    M_KRONOTECH_SRL : UINT := 814; (* Manufacturer: Kronotech Srl (formerly Soltec Soluzioni Tecnologiche Srl) | Location: Basaldella *)
    M_FLIR_SYSTEMS : UINT := 815; (* Manufacturer: FLIR Systems, Inc. | Location: Wilsonville, OR USA - 2017-04-21 *)
    M_UNISTRONG : UINT := 816; (* Manufacturer: UniStrong | Location: Beijing, China - 2017-04-21 *)
    M_TE_CONNECTIVITY_SENSOR_SOLUTIONS : UINT := 817; (* Manufacturer: TE Connectivity Sensor Solutions | Location: Dormund, Germany - 2017-04-21 *)
    M_HGNSS : UINT := 818; (* Manufacturer: HGNSS | Location: Scottsdale, AZ USA - 2017-04-21 *)
    M_PRECO_ELECTRONICS : UINT := 819; (* Manufacturer: Preco Electronics | Location: Boise, ID USA - 2017-04-30 *)
    M_DIALOGIKA_GESELLSCHAFT_FUER_ANGEWANDTE_INFORMATIK_MBH : UINT := 820; (* Manufacturer: DIaLOGIKa Gesellschaft fuer angewandte Informatik mbH | Location: Saarbruecken, *)
    M_THORSEN_TEKNIK : UINT := 821; (* Manufacturer: Thorsen Teknik A/S | Location: Farsø, Denmark - 2017-05-01 *)
    M_BREN_TRONICS : UINT := 822; (* Manufacturer: Bren-Tronics, Inc. | Location: Commack, NY USA - 2017-05-04 *)
    M_ACEINNA : UINT := 823; (* Manufacturer: ACEINNA, Inc (formerly MEMSIC, Inc) | Location: Andover, MA USA - 2017-09-03 *)
    M_UNDHEIM_SYSTEMS : UINT := 824; (* Manufacturer: Undheim Systems AS | Location: Egersund, Norway - 2017-05-04 *)
    M_BPW_HUNG_RIA : UINT := 825; (* Manufacturer: BPW Hungária | Location: Szombathely, Hungary - 2017-05-04 *)
    M_LEWMAR_MARINE : UINT := 826; (* Manufacturer: Lewmar Marine Inc | Location: Guilford, CT USA - 2017-05-05 *)
    M_INMATIX_TECHNOLOGY_GROUP : UINT := 827; (* Manufacturer: INmatix Technology Group Ltd | Location: Hattem, The Netherlands - 2017-05-11 *)
    M_AGRIBRINK : UINT := 828; (* Manufacturer: AgriBrink Inc. | Location: Moorefield, ON Canada - 2017-05-21 *)
    M_DROV_TECHNOLOGIES : UINT := 829; (* Manufacturer: Drov Technologies, Inc. | Location: Oklahoma City, OK USA - 2017-05-22 *)
    M_ULTRA_MOTION : UINT := 830; (* Manufacturer: Ultra Motion LLC | Location: Cutchogue, NY USA - 2017-05-22 *)
    M_DOK_ING : UINT := 831; (* Manufacturer: DOK-ING Ltd. | Location: Zagreb, Croatia - 2017-05-22 *)
    M_HEIZOMAT_GER_TEBAU_ENERGIESYSTEME : UINT := 832; (* Manufacturer: Heizomat Gerätebau-Energiesysteme GmbH | Location: Gunzenhausen, Germany - *)
    M_ELECTRUM_AUTOMATION : UINT := 833; (* Manufacturer: Electrum Automation AB | Location: Umeå, Sweden - 2017-05-24 *)
    M_PIONEER_MICROSYSTEMS : UINT := 834; (* Manufacturer: Pioneer Microsystems, Inc. | Location: Pittsburgh, PA USA - 2017-05-24 *)
    M_PETTRACK : UINT := 835; (* Manufacturer: PetTrack Ltd. | Location: Héreg, Hungary - 2017-05-31 *)
    M_SIGNATURE4 : UINT := 836; (* Manufacturer: Signature4 | Location: Coldwater, OH USA - 2017-05-31 *)
    M_FAMIC_TECHNOLOGIES : UINT := 837; (* Manufacturer: Famic Technologies Inc. | Location: Montréal, QC Canada - 2017-06-11 *)
    M_TEAMSURV : UINT := 838; (* Manufacturer: Teamsurv Ltd | Location: Didcot, Oxfordshire UK - 2017-06-12 *)
    M_INDEXATOR_ROTATOR_SYSTEMS : UINT := 839; (* Manufacturer: Indexator Rotator Systems AB | Location: Vindeln, Sweden - 2017-06-27 *)
    M_E_S_T_E_SRL : UINT := 840; (* Manufacturer: E.S.T.E. srl | Location: Ferrara, Italy - 2017-07-14 *)
    M_AGRA_GPS : UINT := 841; (* Manufacturer: Agra-GPS | Location: Stony Plain, AB Canada - 2017-07-14 *)
    M_DIGIDEVICE_SRL : UINT := 842; (* Manufacturer: DigiDevice Srl | Location: Calvisano, Italy - 2017-07-14 *)
    M_HENDRICKSON_TRUCK_COMMERCIAL_VEHICLE_SYSTEMS : UINT := 843; (* Manufacturer: Hendrickson Truck Commercial Vehicle Systems | Location: Woodridge, IL USA - *)
    M_FELL : UINT := 844; (* Manufacturer: FELL AS | Location: Lier, Norway - 2017-07-14 *)
    M_GMB_G_STROWER_MASCHINENBAU : UINT := 845; (* Manufacturer: GMB Güstrower Maschinenbau GmbH | Location: Güstrow, Germany - 2017-07-16 *)
    M_L3_MAGNET_MOTOR : UINT := 846; (* Manufacturer: L3 Magnet-Motor | Location: Starnberg, Germany - 2017-07-19 *)
    M_OCEANVOLT : UINT := 847; (* Manufacturer: Oceanvolt | Location: Vantaa, Finland - 2017-07-26 *)
    M_NINGUPEX : UINT := 848; (* Manufacturer: ningupex | Location: Dresden, Germany - 2017-07-31 *)
    M_MTS_MASCHINENTECHNIK_SCHRODE_AG : UINT := 849; (* Manufacturer: MTS Maschinentechnik Schrode AG | Location: Hayingen, Germany - 2017-08-06 *)
    M_GEOPROSPECTORS : UINT := 850; (* Manufacturer: Geoprospectors GmbH | Location: Traiskirchen, Austria - 2017-08-08 *)
    M_NOVOTECHNIK_MESSWERTAUFNEHMER_OHG : UINT := 851; (* Manufacturer: Novotechnik Messwertaufnehmer OHG | Location: Ostfildern (Ruit), Germany - *)
    M_VELVAC : UINT := 852; (* Manufacturer: Velvac Inc | Location: New Berlin, WI USA - 2017-08-24 *)
    M_TELEDYNE_RESON_B_V : UINT := 853; (* Manufacturer: Teledyne RESON B.V. | Location: Rotterdam, The Netherlands - 2017-09-05 *)
    M_GEMAC_CHEMNITZ : UINT := 854; (* Manufacturer: GEMAC Chemnitz GmbH | Location: Chemnitz, Germany - 2017-09-05 *)
    M_TOSHIBA_INFRASTRUCTURE_SYSTEMS_AND_SOLUTIONS : UINT := 855; (* Manufacturer: Toshiba Infrastructure Systems & Solutions Corporation | Location: Kawasaki, Japan *)
    M_FARMFACTS : UINT := 856; (* Manufacturer: FarmFacts GmbH | Location: Pfarrkirchen, Germany - 2017-09-10 *)
    M_ZOOMLION_HEAVY_INDUSTRY_NA : UINT := 857; (* Manufacturer: Zoomlion Heavy Industry NA, Inc | Location: Yorkville, WI USA - 2017-09-23 *)
    M_LITTELFUSE : UINT := 858; (* Manufacturer: Littelfuse | Location: Kaunas, Lithuania - 2017-09-23 *)
    M_VALOR : UINT := 859; (* Manufacturer: Valor | Location: Burlington, ON Canada - 2017-09-23 *)
    M_MICHELIN : UINT := 860; (* Manufacturer: Michelin | Location: Clermont-Ferrand, France - 2017-09-27 *)
    M_ADEL_SYSTEM_S_R_L : UINT := 861; (* Manufacturer: Adel System S.r.l. | Location: Reggio Emilia, Italy - 2017-09-27 *)
    M_PROSPEC_ELECTRONICS : UINT := 862; (* Manufacturer: Prospec Electronics | Location: Mount Pleasant, SC USA - 2017-10-20 *)
    M_SMAG : UINT := 863; (* Manufacturer: SMAG | Location: Châlons-en-Champagne, France - 2017-10-20 *)
    M_STREAMLINE_TRANSPORTATION_TECHNOLOGIES : UINT := 864; (* Manufacturer: Streamline Transportation Technologies Inc. | Location: Kamloops, BC Canada - *)
    M_MYEASYFARM : UINT := 865; (* Manufacturer: MyEasyFarm | Location: Prunay, France - 2017-10-20 *)
    M_NETRADYNE : UINT := 866; (* Manufacturer: Netradyne, Inc. | Location: San Diego, CA USA - 2017-10-30 *)
    M_SKELETON_TECHNOLOGIES : UINT := 867; (* Manufacturer: Skeleton Technologies | Location: Lubja, Estonia - 2017-11-03 *)
    M_DATA_PANEL_868 : UINT := 868; (* Manufacturer: Data Panel Corp | Location: Plymouth, MN USA - 2017-11-06 *)
    M_INTERCOMP : UINT := 869; (* Manufacturer: Intercomp | Location: Medina, MN USA - 2017-11-13 *)
    M_TEXTRON_FLEET_MANAGEMENT : UINT := 870; (* Manufacturer: Textron Fleet Management | Location: Surrey, BC Canada - 2017-11-13 *)
    M_AGRI_FAB : UINT := 871; (* Manufacturer: Agri-Fab (formerly Superior Tech Inc) | Location: Sullivan, IL USA - 2021-12-09 *)
    M_K_HLIG_ANTRIEBSTECHNIK : UINT := 872; (* Manufacturer: Kählig Antriebstechnik GmbH | Location: Hannover, Germany - 2017-11-17 *)
    M_GARNET_INSTRUMENTS : UINT := 873; (* Manufacturer: Garnet Instruments Ltd. | Location: Sherwood Park, AB Canada - 2017-12-04 *)
    M_MTA : UINT := 874; (* Manufacturer: MTA S.p.A. | Location: Codogno, Italy - 2017-12-04 *)
    M_SALVARANI_S_R_L : UINT := 875; (* Manufacturer: Salvarani S.r.l. | Location: Poviglio (RE), Italy - 2017-12-04 *)
    M_SUCO_ROBERT_SCHEUFFELE_AND : UINT := 876; (* Manufacturer: SUCO Robert Scheuffele GmbH & Co. KG | Location: Bietigheim-Bissingen, Germany - *)
    M_SICK_ATECH : UINT := 877; (* Manufacturer: SICK ATech GmbH | Location: Witten, Germany - 2017-12-13 *)
    M_FOTON : UINT := 878; (* Manufacturer: FOTON | Location: Beijing, China - 2017-12-13 *)
    M_PG_TRIONIC : UINT := 879; (* Manufacturer: PG Trionic, Inc. | Location: Essex, MA USA - 2017-12-13 *)
    M_REVISION_MILITARY : UINT := 880; (* Manufacturer: Revision Military | Location: Ottawa, ON Canada - 2018-01-08 *)
    M_SOVEMA : UINT := 881; (* Manufacturer: Sovema | Location: Gaggio di Piano, Italy - 2018-01-08 *)
    M_BHTRONIK_AND : UINT := 882; (* Manufacturer: BHTronik GmbH & Co. KG | Location: Oberviechtach, Germany - 2018-01-08 *)
    M_SWIFT_NAVIGATION : UINT := 883; (* Manufacturer: Swift Navigation, Inc. | Location: San Francisco, CA USA - 2018-01-08 *)
    M_SURE_GRIP_CONTROLS : UINT := 884; (* Manufacturer: Sure Grip Controls Inc. | Location: Saanichton, BC Canada - 2018-01-09 *)
    M_SICK_AG : UINT := 885; (* Manufacturer: SICK AG (formerly SICK Stegmann GmbH) | Location: Donaueschingen, Germany - *)
    M_HITACHI_ZOSEN : UINT := 886; (* Manufacturer: Hitachi Zosen Corporation | Location: Osaka, Japan - 2018-01-23 *)
    M_TURNTIDE_TRANSPORT_LIMITED_887 : UINT := 887; (* Manufacturer: Turntide Transport Limited (formerly Hyperdrive Innovation Limited) | Location: *)
    M_CARMA_SYSTEMS : UINT := 888; (* Manufacturer: Carma Systems Inc | Location: Albany, NY USA - 2018-01-23 *)
    M_SANY_AMERICA : UINT := 889; (* Manufacturer: SANY America Inc | Location: Peachtree City, GA USA - 2018-01-23 *)
    M_L3_TECHNOLOGIES : UINT := 890; (* Manufacturer: L3 Technologies, Inc. | Location: Sarasota, FL USA - 2018-01-26 *)
    M_CARRIERWEB : UINT := 891; (* Manufacturer: CarrierWeb | Location: Atlanta, GA USA - 2018-02-01 *)
    M_MECTRONX : UINT := 892; (* Manufacturer: Mectronx Corp | Location: Sun Prairie, WI USA - 2018-02-04 *)
    M_KLINKTECHNICS : UINT := 893; (* Manufacturer: KlinkTechnics Ltd. | Location: Beaver Dam, WI USA - 2018-02-07 *)
    M_RHODAN_MARINE_SYSTEMS_OF_FLORIDA : UINT := 894; (* Manufacturer: Rhodan Marine Systems of Florida LLC (Duplicate entry; use MFR ID 1012) | Location: *)
    M_PELOTON_TECHNOLOGY : UINT := 895; (* Manufacturer: Peloton Technology | Location: Mountain View, CA USA - 2018-02-10 *)
    M_NEXTFOUR_SOLUTIONS : UINT := 896; (* Manufacturer: NextFour Solutions Ltd | Location: Turku, Finland - 2018-02-10 *)
    M_DOT_TECHNOLOGY : UINT := 897; (* Manufacturer: Dot Technology Corp. | Location: Emerald Park, SK Canada - 2018-02-14 *)
    M_JOSEF_KOTTE_LANDTECHNIK_AND : UINT := 898; (* Manufacturer: Josef Kotte Landtechnik GmbH & Co. KG | Location: Rieste, Germany - 2018-02-20 *)
    M_LIPPERT_COMPONENTS : UINT := 899; (* Manufacturer: Lippert Components, Inc | Location: Sterling Heights, MI USA - 2018-03-04 *)
    M_OSB_CONNAGTIVE : UINT := 900; (* Manufacturer: OSB connagtive GmbH (formerly OSB AG) | Location: Munich, Germany - 2021-08-03 *)
    M_ZIVAN_SRL : UINT := 901; (* Manufacturer: Zivan Srl | Location: Poviglio, Italy - 2018-03-04 *)
    M_BUCHER_HYDRAULICS : UINT := 902; (* Manufacturer: Bucher Hydraulics | Location: Neuheim, Switzerland - 2018-03-04 *)
    M_INMOTION : UINT := 903; (* Manufacturer: InMotion | Location: Blacksburg, VA USA - 2018-03-08 *)
    M_EQUIPMENT_SAFETY_SYSTEMS_PTY : UINT := 904; (* Manufacturer: Equipment Safety Systems Pty. Ltd. (EQSS) | Location: Seaford, Victoria Australia - *)
    M_ASA_ELECTRONICS_905 : UINT := 905; (* Manufacturer: ASA Electronics | Location: Elkhart, IN USA - 2018-03-15 *)
    M_MOBA_AG : UINT := 906; (* Manufacturer: MOBA AG | Location: Limburg, Germany - 2018-04-25 *)
    M_STRAUTMANN : UINT := 907; (* Manufacturer: strautmann | Location: Bad Laer, Germany - 2018-04-15 *)
    M_CHONBUK_NATIONAL_UNIVERSITY_DEPARTMENT_OF_ELECTRONICS : UINT := 908; (* Manufacturer: Chonbuk National University Department of Electronics | Location: Jeonju, Republic *)
    M_MARINES : UINT := 909; (* Manufacturer: Marines Co., Ltd. | Location: Ulsan, Republic of Korea - 2018-04-17 *)
    M_HERMANN_PAUS_MASCHINENFABRIK : UINT := 910; (* Manufacturer: Hermann Paus Maschinenfabrik GmbH | Location: Emsbüren, Germany - 2018-04-25 *)
    M_NAUTIC_ON : UINT := 911; (* Manufacturer: Nautic-On | Location: Chicago, IL USA - 2018-04-25 *)
    M_STEYR_MOTORS : UINT := 912; (* Manufacturer: Steyr Motors GmbH | Location: Steyr, Austria - 2018-04-25 *)
    M_TOYOTA_MOTOR : UINT := 913; (* Manufacturer: Toyota Motor Corporation | Location: Toyota City, Japan - 2018-04-25 *)
    M_ZETOR_TRACTORS_A_S : UINT := 914; (* Manufacturer: ZETOR TRACTORS a.s. | Location: Brno, Czech Republic - 2018-05-07 *)
    M_DOSIFICACION_Y_SISTEMAS_ELECTRONICOS_S_L : UINT := 915; (* Manufacturer: Dosificacion y sistemas electronicos S.L. (DSE) | Location: Mieres, Spain - *)
    M_HANS_TURCK_AND : UINT := 916; (* Manufacturer: Hans Turck GmbH & Co. KG (formerly Turck Inc.) | Location: Mülheim an der Ruhr, *)
    M_SENTINEL_D_O_O : UINT := 917; (* Manufacturer: Sentinel d.o.o. | Location: Vodnjan, Crotia - 2018-05-13 *)
    M_AMW_MACHINE_CONTROL : UINT := 918; (* Manufacturer: AMW Machine Control, Inc | Location: Saranac, MI USA - 2018-05-16 *)
    M_FURRION : UINT := 919; (* Manufacturer: Furrion LLC | Location: Elkhart, IN USA - 2018-05-16 *)
    M_MTD_CONSUMER_GROUP : UINT := 920; (* Manufacturer: MTD Consumer Group Inc. | Location: Valley City, OH USA - 2018-05-18 *)
    M_ROPA_FAHRZEUG_UND_MASCHINENBAU : UINT := 921; (* Manufacturer: ROPA Fahrzeug- und Maschinenbau GmbH | Location: Herrngiersdorf, Germany - *)
    M_TERBERG_BENSCHOP_B_V : UINT := 922; (* Manufacturer: Terberg Benschop B.V. | Location: Benschop, The Netherlands - 2018-05-25 *)
    M_ELTEK : UINT := 923; (* Manufacturer: ELTEK S.p.A. | Location: Casale Monferrato, Italy - 2018-06-03 *)
    M_PAS_PESCHAK_AUTONOME_SYSTEME : UINT := 924; (* Manufacturer: PAS Peschak Autonome Systeme GmbH | Location: Großweikersdorf, Austria - 2018-06-03 *)
    M_GW_LISK_COMPANY : UINT := 925; (* Manufacturer: GW Lisk Company | Location: Clifton Springs, NY USA - 2018-06-03 *)
    M_BUHLER_INDUSTRIES : UINT := 926; (* Manufacturer: Buhler Industries Inc. | Location: Winnipeg, MB Canada - 2018-06-03 *)
    M_SAICON : UINT := 927; (* Manufacturer: Saicon | Location: Passo Fundo, Brazil - 2018-06-03 *)
    M_EAO_AUTOMOTIVE_AND : UINT := 928; (* Manufacturer: EAO Automotive GmbH & Co. KG | Location: Auerbach, Germany - 2018-06-05 *)
    M_JL_MARINE_SYSTEMS : UINT := 929; (* Manufacturer: Jl Marine Systems, Inc. | Location: Tampa, FL USA - 2018-06-07 *)
    M_ECOTRONIX : UINT := 930; (* Manufacturer: Ecotronix Corp. | Location: Seoul, Republic of Korea - 2018-06-07 *)
    M_ENERTEC_MARINE : UINT := 931; (* Manufacturer: Enertec Marine Ltd | Location: Auckland, New Zealand - 2018-06-14 *)
    M_DISCOVER_BATTERY : UINT := 932; (* Manufacturer: Discover Battery | Location: Richmond, BC Canada - 2018-06-25 *)
    M_DELTA_MOBILE_SYSTEMS : UINT := 933; (* Manufacturer: Delta Mobile Systems, Inc. | Location: Elgin, IL USA - 2018-06-25 *)
    M_FARMOBILE : UINT := 934; (* Manufacturer: Farmobile, Inc. | Location: Leawood, KS USA - 2018-06-25 *)
    M_MEELS_AND : UINT := 935; (* Manufacturer: Meels GmbH & Co. KG | Location: Fellheim, Germany - 2018-06-29 *)
    M_HI_TECH_MILLENNIUM : UINT := 936; (* Manufacturer: Hi-tech Millennium | Location: Corunna, MI, USA - 2018-06-29 *)
    M_PRECISION_CIRCUITS : UINT := 937; (* Manufacturer: Precision Circuits Inc | Location: Downers Grove, IL USA - 2018-06-29 *)
    M_LEVEL_SYSTEMS : UINT := 938; (* Manufacturer: LEVEL Systems | Location: Náchod, Czech Republic - 2018-06-29 *)
    M_WARN_INDUSTRIES : UINT := 939; (* Manufacturer: Warn Industries, Inc. | Location: Clackamas, OR USA - 2018-06-29 *)
    M_DOMETAL_OY : UINT := 940; (* Manufacturer: Dometal Oy | Location: Loimaa, Finland - 2018-06-29 *)
    M_NAVYA : UINT := 941; (* Manufacturer: Navya | Location: Villeurbanne, France - 2018-06-29 *)
    M_VOGELSANG_AND : UINT := 942; (* Manufacturer: Vogelsang GmbH & Co. KG | Location: Essen, Germany - 2018-07-08 *)
    M_FISCHER_AG_PR_ZISIONSPINDELN : UINT := 943; (* Manufacturer: FISCHER AG Präzisionspindeln | Location: Herzogenbuchsee, Switzerland - 2018-07-08 *)
    M_ZONTISA_MARINE_SL : UINT := 944; (* Manufacturer: ZONTISA Marine SL | Location: Barcelona, Spain - 2018-07-08 *)
    M_EQUALIZER_AG : UINT := 945; (* Manufacturer: Equalizer AG | Location: Cape Town, South Africa - 2018-07-13 *)
    M_HYDAC_TECNOLOGIA_LTDA : UINT := 946; (* Manufacturer: Hydac Tecnologia Ltda | Location: São Bernardo do Campo, Brazil - 2018-07-13 *)
    M_GERD_B_R : UINT := 947; (* Manufacturer: Gerd Bär GmbH | Location: Heilbronn, Germany - 2018-07-21 *)
    M_DONIX : UINT := 948; (* Manufacturer: Donix | Location: Cape Town, South Africa - 2018-07-21 *)
    M_KODA_ELECTRIC_A_S : UINT := 949; (* Manufacturer: Škoda Electric a.s. | Location: Plzeň, Czech Republic - 2018-07-25 *)
    M_RE_LAB_S_R_L : UINT := 950; (* Manufacturer: RE:Lab s.r.l. | Location: Reggio Emilia, Italy - 2018-08-01 *)
    M_EXOR_INTERNATIONAL : UINT := 951; (* Manufacturer: Exor International S.p.A. | Location: San Giovanni Lupatoto, Italy - 2018-08-06 *)
    M_TAN_DELTA_SYSTEMS : UINT := 952; (* Manufacturer: Tan Delta Systems Ltd | Location: Sheffield, South Yorkshire UK - 2018-08-24 *)
    M_CURTISS_WRIGHT : UINT := 953; (* Manufacturer: Curtiss-Wright | Location: Davidson, NC USA - 2018-08-30 *)
    M_SETEC_PTY : UINT := 954; (* Manufacturer: Setec Pty Ltd | Location: Melbourne, Victoria Australia - 2018-08-30 *)
    M_HOTTINGER_BALDWIN_ELECTRONIC_MEASUREMENT_TECHNOLOGY : UINT := 955; (* Manufacturer: Hottinger Baldwin (Suzhou) Electronic Measurement Technology Co., Ltd. | Location: *)
    M_PIHER_SENSORS_AND_CONTROLS : UINT := 956; (* Manufacturer: Piher Sensors & Controls S.A. | Location: Tudela, Spain - 2018-09-08 *)
    M_SIERRA_WIRELESS : UINT := 957; (* Manufacturer: Sierra Wireless Inc | Location: Richmond, BC Canada - 2018-09-08 *)
    M_NHK_MEC : UINT := 958; (* Manufacturer: NHK MEC Corporation | Location: Yokohama, Japan - 2018-09-08 *)
    M_CASCADE : UINT := 959; (* Manufacturer: Cascade Corporation | Location: Fairview, OR USA - 2018-09-21 *)
    M_VEMCON : UINT := 960; (* Manufacturer: Vemcon GmbH | Location: Munich, Germany - 2018-09-21 *)
    M_POK_SAS : UINT := 961; (* Manufacturer: POK SAS | Location: Nogent-sur-Seine, France - 2018-10-03 *)
    M_TIMBOLIER_INDUSTRIES : UINT := 962; (* Manufacturer: Timbolier Industries, Inc. | Location: Edgewater, MD USA - 2018-10-03 *)
    M_THOMASON_JONES_COMPANY : UINT := 963; (* Manufacturer: Thomason Jones Company, LLC | Location: Anacortes, WA USA - 2018-10-05 *)
    M_AGROVIR_KFT : UINT := 964; (* Manufacturer: AgroVIR Kft | Location: Tata, Hungary - 2018-10-05 *)
    M_RO_SYS_SOFTWARE : UINT := 965; (* Manufacturer: Ro-Sys Software | Location: Debrecen, Hungary - 2018-10-05 *)
    M_VISIBLEFARM : UINT := 966; (* Manufacturer: VisibleFarm | Location: Tata, Hungary - 2018-10-05 *)
    M_MOTECK_ELECTRIC : UINT := 967; (* Manufacturer: Moteck Electric Corp. | Location: New Taipei City, Taiwan - 2018-10-21 *)
    M_COX_POWERTRAIN_LIMITED : UINT := 968; (* Manufacturer: Cox Powertrain Limited | Location: Shoreham-by-Sea, West Sussex UK - 2018-10-24 *)
    M_BLUE_SEA_SYSTEMS : UINT := 969; (* Manufacturer: Blue Sea Systems | Location: Bellingham, WA USA - 2018-10-24 *)
    M_JABONI_POWER_PRODUCTS : UINT := 970; (* Manufacturer: Jaboni Power Products, LLC | Location: Elkhart, IN USA - 2018-10-27 *)
    M_B_B_SMARTWORX : UINT := 971; (* Manufacturer: B+B Smartworx | Location: Ottawa, IL USA - 2018-11-06 *)
    M_AXION_AG : UINT := 972; (* Manufacturer: Axion AG | Location: Weissenhorn, Germany - 2018-11-19 *)
    M_ZASSO : UINT := 973; (* Manufacturer: Zasso GmbH | Location: Aachen, Germany - 2018-11-19 *)
    M_PICO_TECHNOLOGY_LIMITED : UINT := 974; (* Manufacturer: Pico Technology Limited | Location: St. Neots, Cambridgeshire UK - 2018-12-10 *)
    M_SIEMENS_AG : UINT := 975; (* Manufacturer: Siemens AG | Location: Fuerth, Germany - 2018-12-10 *)
    M_DERIVE_SYSTEMS : UINT := 976; (* Manufacturer: Derive Systems, Inc. | Location: Sanford, FL USA - 2018-12-11 *)
    M_COPELAND_LP : UINT := 977; (* Manufacturer: Copeland LP (formerly Emerson Electric Co.) | Location: St. Louis, MO USA - *)
    M_CANFIELD_CONNECTOR : UINT := 978; (* Manufacturer: Canfield Connector | Location: Youngstown, OH USA - 2018-12-18 *)
    M_MCHALE : UINT := 979; (* Manufacturer: McHale | Location: Ballinrobe, Ireland - 2018-12-18 *)
    M_GUSSI_ITALIA_S_R_L : UINT := 980; (* Manufacturer: Gussi Italia S.R.L. | Location: Tregnago, Italy - 2018-12-18 *)
    M_KOBELT_MANUFACTURING : UINT := 981; (* Manufacturer: Kobelt Manufacturing Co. Ltd | Location: Surrey, BC Canada - 2018-12-18 *)
    M_BRIGGS_AND_STRATTON : UINT := 982; (* Manufacturer: Briggs & Stratton Corporation | Location: Wauwatosa, WI USA - 2018-12-20 *)
    M_DEZWAEF_NV : UINT := 983; (* Manufacturer: Dezwaef NV | Location: Moerkerke, Belgium - 2019-01-04 *)
    M_E_T_A_ELEKTROTECHNISCHE_APPARATE : UINT := 984; (* Manufacturer: E-T-A Elektrotechnische Apparate GmbH | Location: Altdorf, Germany - 2019-01-04 *)
    M_NLR : UINT := 985; (* Manufacturer: NLR, LLC | Location: Opelika, AL USA - 2019-02-03 *)
    M_AAMP_GLOBAL : UINT := 986; (* Manufacturer: AAMP Global | Location: Bordon, Hampshire UK - 2019-02-08 *)
    M_BALTIC_CAR_EQUIPMENT : UINT := 987; (* Manufacturer: Baltic Car Equipment | Location: Kaunas, Lithuania - 2019-02-08 *)
    M_VOITH_TURBO : UINT := 988; (* Manufacturer: Voith Turbo | Location: Heidenheim, Germany - 2019-02-08 *)
    M_FLUX_GER_TE : UINT := 989; (* Manufacturer: Flux-Geräte GmbH | Location: Maulbronn, Germany - 2019-02-13 *)
    M_SAMSUNG_SDI : UINT := 990; (* Manufacturer: SAMSUNG SDI Co., Ltd. | Location: Cheonan, Republic of Korea - 2019-02-20 *)
    M_DEUTRONIC_ELEKTRONIK : UINT := 991; (* Manufacturer: Deutronic Elektronik GmbH | Location: Adlkofen, Germany - 2019-02-28 *)
    M_MARINEIOT : UINT := 992; (* Manufacturer: MarineIOT LLC | Location: Seattle, WA USA - 2019-03-06 *)
    M_ALELION_ENERGY_SYSTEMS : UINT := 993; (* Manufacturer: Alelion Energy Systems AB | Location: Gothenburg, Sweden - 2019-03-10 *)
    M_MORRIS_INDUSTRIES : UINT := 994; (* Manufacturer: Morris Industries Ltd. | Location: Saskatoon, SK Canada - 2019-03-14 *)
    M_CIRCUITLINK_PTY : UINT := 995; (* Manufacturer: Circuitlink Pty Ltd. | Location: Seven Hills, NSW Australia - 2019-03-14 *)
    M_ENIQUEST_PTY : UINT := 996; (* Manufacturer: Eniquest Pty Ltd | Location: Bells Creek, QLD Australia - 2019-03-26 *)
    M_XENTA_SYSTEMS_SRL : UINT := 997; (* Manufacturer: Xenta Systems Srl | Location: Rome, Italy - 2019-03-26 *)
    M_TRANSCELL_TECHNOLOGY : UINT := 998; (* Manufacturer: Transcell Technology Inc | Location: Buffalo Grove, IL USA - 2019-04-02 *)
    M_TERRATRONIQ_B_V : UINT := 999; (* Manufacturer: TerraTroniq B.V. | Location: Renkum, The Netherlands - 2019-04-02 *)
    M_LANDMASCHINEN_WIENHOFF : UINT := 1000; (* Manufacturer: Landmaschinen Wienhoff GmbH | Location: Bawinkel, Germany - 2019-04-11 *)
    M_CLERAL : UINT := 1001; (* Manufacturer: Cleral Inc. | Location: Val-d'Or, QC Canada - 2019-04-19 *)
    M_KUSSMAUL_ELECTRONICS : UINT := 1002; (* Manufacturer: Kussmaul Electronics Co. | Location: West Sayville, NY USA - 2019-04-19 *)
    M_TECHNOTRANS_SE : UINT := 1003; (* Manufacturer: technotrans SE | Location: Sassenberg, Germany - 2019-04-19 *)
    M_ULTRAFLEX : UINT := 1004; (* Manufacturer: Ultraflex SpA | Location: Casella, Italy - 2019-04-19 *)
    M_TSE_BRAKES : UINT := 1005; (* Manufacturer: TSE Brakes, Inc. | Location: Cullman, AL USA - 2019-04-19 *)
    M_PROTERRA : UINT := 1006; (* Manufacturer: Proterra | Location: Burlingame, CA USA - 2019-04-29 *)
    M_MASCHINENFABRIK_MEYER_LOHNE : UINT := 1007; (* Manufacturer: Maschinenfabrik Meyer-Lohne GmbH | Location: Lohne, Germany - 2019-04-29 *)
    M_LINTEST_SYSTEMS : UINT := 1008; (* Manufacturer: Lintest Systems LLC | Location: Boca Raton, FL USA - 2019-04-29 *)
    M_TOUCHTRONICS : UINT := 1009; (* Manufacturer: TouchTronics, Inc. | Location: Elkhart, IN USA - 2019-05-03 *)
    M_AGRICULTURAL_INDUSTRY_ELECTRONICS_FOUNDATION_E_V : UINT := 1010; (* Manufacturer: Agricultural Industry Electronics Foundation e.V. | Location: Frankfurt, Germany - *)
    M_SOUNDMAX_ELECTRONICS : UINT := 1011; (* Manufacturer: Soundmax Electronics Ltd | Location: Hong Kong, China - 2019-05-07 *)
    M_RHODAN_MARINE_SYSTEMS_OF_FLORIDA_1012 : UINT := 1012; (* Manufacturer: Rhodan Marine Systems of Florida LLC | Location: Sarasota, FL USA - 2019-05-15 *)
    M_ALLOCHIS_E_TEC : UINT := 1013; (* Manufacturer: Allochis E-Tec | Location: Ferré, Argentina - 2019-05-24 *)
    M_BRIRI_MASCHINENBAU : UINT := 1014; (* Manufacturer: Briri Maschinenbau GmbH | Location: Bawinkel, Germany - 2019-05-24 *)
    M_SECURITAG_SAS : UINT := 1015; (* Manufacturer: SECURITAG SAS | Location: Nantes, France - 2019-05-24 *)
    M_R_HREN_UND_PUMPENWERK_BAUER : UINT := 1016; (* Manufacturer: Röhren- und Pumpenwerk BAUER GmbH | Location: Voitsberg, Austria - 2019-06-14 *)
    M_CALDARO : UINT := 1017; (* Manufacturer: Caldaro AB | Location: Stockholm, Sweden - 2019-06-14 *)
    M_FLEX_TTS : UINT := 1018; (* Manufacturer: Flex TTS | Location: San Jose, CA USA - 2019-06-14 *)
    M_CODEK_FOUNDRIES : UINT := 1019; (* Manufacturer: Codek Foundries | Location: Cedar Rapids, IA USA - 2019-06-14 *)
    M_ONYX_MARINE_AUTOMATION_S_R_L : UINT := 1020; (* Manufacturer: Onyx Marine Automation s.r.l. | Location: Fano, Italy - 2019-06-14 *)
    M_ENTRATECH_SYSTEMS : UINT := 1021; (* Manufacturer: Entratech Systems LLC | Location: Sandusky, OH USA - 2019-06-14 *)
    M_ITC : UINT := 1022; (* Manufacturer: ITC Inc | Location: Hudsonville, MI USA - 2019-06-14 *)
    M_PEAK_SYSTEM_TECHNIK : UINT := 1023; (* Manufacturer: PEAK-System Technik GmbH | Location: Darmstadt, Germany - 2019-06-21 *)
    M_INVENTUS_POWER : UINT := 1024; (* Manufacturer: Inventus Power | Location: Woodridge, IL USA - 2019-06-21 *)
    M_EZE_SYSTEM : UINT := 1025; (* Manufacturer: eze System, Inc. | Location: Folsom, CA USA - 2019-06-25 *)
    M_ZTR_CONTROL_SYSTEMS : UINT := 1026; (* Manufacturer: ZTR Control Systems, LLC | Location: London, ON Canada - 2019-06-25 *)
    M_GOLDACRES_PTY : UINT := 1027; (* Manufacturer: Goldacres PTY LTD | Location: Mitchell Park, Victoria Australia - 2019-06-25 *)
    M_AUTEL_INTELLIGENT_TECHNOLOGY : UINT := 1028; (* Manufacturer: Autel Intelligent Technology Corp., Ltd | Location: Shenzhen, China - 2019-06-29 *)
    M_THE_MARINE_GUARDIAN : UINT := 1029; (* Manufacturer: The Marine Guardian LLC | Location: Spring Hill, FL USA - 2019-06-29 *)
    M_TUME_AGRI_OY : UINT := 1030; (* Manufacturer: Tume-Agri Oy | Location: Turenki, Finland - 2019-07-11 *)
    M_FLINTEC_UK : UINT := 1031; (* Manufacturer: Flintec UK Ltd. | Location: Cardiff, UK - 2019-07-22 *)
    M_SIMOL : UINT := 1032; (* Manufacturer: SIMOL S.p.A. | Location: Codisotto (RE), Italy - 2019-07-22 *)
    M_ECCO_SAFETY_GROUP : UINT := 1033; (* Manufacturer: ECCO Safety Group | Location: Boise, ID USA - 2019-08-02 *)
    M_SIREN_MARINE : UINT := 1034; (* Manufacturer: Siren Marine | Location: Newport, RI USA - 2019-08-02 *)
    M_AGRES : UINT := 1035; (* Manufacturer: Agres | Location: Pinhais, Brazil - 2019-08-16 *)
    M_BENDER_AND : UINT := 1036; (* Manufacturer: Bender GmbH & Co. KG | Location: Grünberg, Germany - 2019-08-16 *)
    M_DRAGONFLY_ENERGY : UINT := 1037; (* Manufacturer: Dragonfly Energy Corp. | Location: Sparks, NV USA - 2019-08-16 *)
    M_EMIT_TECHNOLOGIES : UINT := 1038; (* Manufacturer: EMIT Technologies, Inc. | Location: Sheridan, WY USA - 2019-08-16 *)
    M_LIUGONG_DRESSTA_MACHINERY : UINT := 1039; (* Manufacturer: Liugong Dressta Machinery | Location: Stalowa Wola, Poland - 2019-08-20 *)
    M_BPE_ELECTRONICS_SRL : UINT := 1040; (* Manufacturer: BPE Electronics Srl | Location: Campagnola Emilia (RE), Italy - 2019-08-28 *)
    M_EZ_LYNK : UINT := 1041; (* Manufacturer: EZ Lynk | Location: Georgetown, Cayman Islands - 2019-08-28 *)
    M_ENGCON_GROUP : UINT := 1042; (* Manufacturer: engcon group | Location: Strömsund, Sweden - 2019-08-28 *)
    M_HYVA : UINT := 1043; (* Manufacturer: Hyva | Location: Alphen Aan Den Rijn, The Netherlands - 2019-09-20 *)
    M_XEE : UINT := 1044; (* Manufacturer: Xee | Location: Lille, France - 2019-09-20 *)
    M_CMR_GROUP : UINT := 1045; (* Manufacturer: CMR Group | Location: Marseille, France - 2019-09-20 *)
    M_PRAXIDYN : UINT := 1046; (* Manufacturer: Praxidyn | Location: Oakland, IA USA - 2019-10-02 *)
    M_SONIC : UINT := 1047; (* Manufacturer: Sonic Corporation | Location: Tokyo, Japan - 2019-10-02 *)
    M_AGRIVATION_UG : UINT := 1048; (* Manufacturer: Agrivation UG | Location: Havixbeck, Germany - 2019-10-02 *)
    M_S_AND_S_CYCLE : UINT := 1049; (* Manufacturer: S&S Cycle | Location: Viola, WI USA - 2019-10-07 *)
    M_SPACENUS : UINT := 1050; (* Manufacturer: Spacenus GmbH | Location: Darmstadt, Germany - 2019-10-07 *)
    M_PRONAV : UINT := 1051; (* Manufacturer: ProNav AS | Location: Egersund, Norway - 2019-10-09 *)
    M_PFREUNDT : UINT := 1052; (* Manufacturer: Pfreundt | Location: Südlohn, Germany - 2019-10-16 *)
    M_VETUS_MAXWELL : UINT := 1053; (* Manufacturer: Vetus Maxwell, Inc. | Location: Hanover, MD USA - 2019-10-16 *)
    M_SCHMOTZER_HACKTECHNIK_AND : UINT := 1054; (* Manufacturer: Schmotzer Hacktechnik GmbH & Co. KG | Location: Bad Windsheim, Germany - 2019-10-24 *)
    M_EXA_COMPUTING : UINT := 1055; (* Manufacturer: EXA Computing GmbH | Location: Hamm, Germany - 2019-10-24 *)
    M_LITHIUM_PROS : UINT := 1056; (* Manufacturer: Lithium Pros | Location: Knoxville, TN USA - 2019-11-05 *)
    M_EQUIPMENTSHARE : UINT := 1057; (* Manufacturer: EquipmentShare | Location: Columbia, MO USA - 2019-11-12 *)
    M_BONDIOLI_AND_PAVESI : UINT := 1058; (* Manufacturer: Bondioli & Pavesi SpA | Location: Pieve di Cento, Italy - 2019-11-12 *)
    M_BOATRAX : UINT := 1059; (* Manufacturer: Boatrax | Location: Miami, FL USA - 2019-11-18 *)
    M_SCALE_TEC : UINT := 1060; (* Manufacturer: Scale-Tec | Location: Anamosa, IA USA - 2019-12-01 *)
    M_VOLVO_CONSTRUCTION_EQUIPMENT : UINT := 1061; (* Manufacturer: Volvo Construction Equipment | Location: Shippensburg, PA USA - 2019-12-01 *)
    M_MAROL : UINT := 1062; (* Manufacturer: Marol Co Ltd | Location: Kobe, Japan - 2019-12-01 *)
    M_SOLSTEER : UINT := 1063; (* Manufacturer: SolSteer | Location: Pulborough, West Sussex UK - 2019-12-01 *)
    M_OMNITECH_ROBOTICS : UINT := 1064; (* Manufacturer: Omnitech Robotics Inc. | Location: Littleton, CO USA - 2019-12-14 *)
    M_CALYPSO_INSTRUMENTS : UINT := 1065; (* Manufacturer: CALYPSO Instruments | Location: Zaragoza, Spain - 2019-12-14 *)
    M_SPOT_ZERO_WATER : UINT := 1066; (* Manufacturer: Spot Zero Water | Location: Fort Lauderdale, FL USA - 2019-12-14 *)
    M_TECOMEC_S_R_L : UINT := 1067; (* Manufacturer: Tecomec S.r.l. | Location: Reggio Emilia (RE), Italy - 2019-12-14 *)
    M_ZAPI : UINT := 1068; (* Manufacturer: Zapi S.p.A. | Location: Poviglio (RE), Italy - 2019-12-14 *)
    M_LITHIONICS_BATTERY : UINT := 1069; (* Manufacturer: Lithionics Battery LLC | Location: Clearwater, FL USA - 2020-01-07 *)
    M_QUICK_TECK_ELECTRONICS : UINT := 1070; (* Manufacturer: Quick-teck Electronics Ltd | Location: Newark Close, Royston UK - 2020-01-07 *)
    M_MACH_SYSTEMS_S_R_O : UINT := 1071; (* Manufacturer: MACH SYSTEMS s.r.o. | Location: Prague, Czech Republic - 2020-01-08 *)
    M_LA_MARCHE_MANUFACTURING_COMPANY : UINT := 1072; (* Manufacturer: La Marche Manufacturing Company | Location: Des Plaines, IA USA - 2020-01-10 *)
    M_MANITOU_EQUIPMENT_AMERICA : UINT := 1073; (* Manufacturer: Manitou Equipment America LLC | Location: West Bend, WI USA - 2020-01-15 *)
    M_KINDHELM_NAVIGS_OY : UINT := 1074; (* Manufacturer: Kindhelm / Navigs Oy | Location: Espoo, Finland - 2020-01-15 *)
    M_UNIDEN_AMERICA : UINT := 1075; (* Manufacturer: Uniden America Corporation | Location: Irving, TX USA - 2020-01-17 *)
    M_DOGA : UINT := 1076; (* Manufacturer: DOGA S.A. | Location: Abrera, Barcelona Spain - 2020-01-17 *)
    M_YMER_TECHNOLOGY : UINT := 1077; (* Manufacturer: Ymer Technology | Location: Stockholm, Sweden - 2020-01-17 *)
    M_GE_APPLIANCES : UINT := 1078; (* Manufacturer: GE Appliances | Location: Louisville, KY USA - 2020-01-25 *)
    M_CARL_ZEISS_SPECTROSCOPY : UINT := 1079; (* Manufacturer: Carl Zeiss Spectroscopy GmbH | Location: Jena, Germany - 2020-01-28 *)
    M_EPSILOR_ELECTRIC_FUEL : UINT := 1080; (* Manufacturer: Epsilor-Electric Fuel Ltd. | Location: Beit Shemesh, Israel - 2020-01-30 *)
    M_IMCON_ELECTRONICS_S_R_O : UINT := 1081; (* Manufacturer: Imcon Electronics, s.r.o. | Location: Šlapanice, Czech Republic - 2020-02-11 *)
    M_T_MOSAN_ENGINE_AND_TRACTOR : UINT := 1082; (* Manufacturer: TÜMOSAN Engine and Tractor Co. | Location: Istanbul, Turkey - 2020-02-11 *)
    M_NAUTICONCEPT : UINT := 1083; (* Manufacturer: Nauticoncept | Location: Macon, France - 2020-02-11 *)
    M_SHADOW_CASTER_LED_LIGHTING : UINT := 1084; (* Manufacturer: Shadow-Caster LED lighting LLC | Location: Clearwater, FL USA - 2020-02-11 *)
    M_WET_SOUNDS : UINT := 1085; (* Manufacturer: Wet Sounds, LLC | Location: Houston, TX USA - 2020-02-21 *)
    M_LIFE_RACING : UINT := 1086; (* Manufacturer: Life Racing Ltd | Location: Basildon, Essex UK - 2020-02-21 *)
    M_ITPHOTONICS_S_R_L : UINT := 1087; (* Manufacturer: ITPhotonics S.r.l. | Location: Fara Vicentino, Italy - 2020-02-21 *)
    M_E_T_A_CIRCUIT_BREAKERS : UINT := 1088; (* Manufacturer: E-T-A Circuit Breakers | Location: Mt. Prospect, IL USA - 2020-02-21 *)
    M_CARROSSERIE_HESS_AG : UINT := 1089; (* Manufacturer: Carrosserie HESS AG | Location: Bellach, Switzerland - 2020-03-03 *)
    M_E_T_A_CIRCUIT_BREAKERS_1090 : UINT := 1090; (* Manufacturer: E-T-A Circuit Breakers Ltd | Location: Aylesbury, Buckinghamshire UK - 2020-03-05 *)
    M_WHEEL_MONITOR : UINT := 1091; (* Manufacturer: Wheel Monitor Inc. | Location: Niagara-on-the-Lake, ON Canada - 2020-03-15 *)
    M_SCHEIBER : UINT := 1092; (* Manufacturer: Scheiber | Location: Saint-Pierre du Chemin, France - 2020-03-24 *)
    M_INNOLECTRIC : UINT := 1093; (* Manufacturer: innolectric | Location: Bochum, Germany - 2020-03-31 *)
    M_TOKUSHU_DENKI : UINT := 1094; (* Manufacturer: Tokushu Denki | Location: Iwata, Japan - 2020-04-17 *)
    M_WEG_DRIVES_AND_CONTROLS_AUTOMA_O_LTDA : UINT := 1095; (* Manufacturer: WEG Drives and Controls - Automação Ltda | Location: Jaraguá do Sul, Brazil - *)
    M_TEXENSE_SENSORS : UINT := 1096; (* Manufacturer: Texense Sensors | Location: Varennes-Vauzelles, France - 2020-04-28 *)
    M_M2M_CRAFT : UINT := 1097; (* Manufacturer: M2M Craft Co., Ltd | Location: Sapporo, Japan - 2020-04-28 *)
    M_PREH : UINT := 1098; (* Manufacturer: Preh GmbH | Location: Bad Neustadt a. d. Saale, Germany - 2020-05-12 *)
    M_MADGETECH : UINT := 1099; (* Manufacturer: MadgeTech, Inc | Location: Warner, NH USA - 2020-05-13 *)
    M_LINK_MARINE_TECHNOLOGIES : UINT := 1100; (* Manufacturer: LINK Marine Technologies (formerly Smart Yachts International Limited) | Location: *)
    M_DIS_SENSORS_B_V : UINT := 1101; (* Manufacturer: DIS Sensors B.V. | Location: Soest, the Netherlands - 2020-06-04 *)
    M_CARL_GERINGHOFF_AND : UINT := 1102; (* Manufacturer: Carl Geringhoff GmbH & Co. KG | Location: Ahlen, Germany - 2020-06-04 *)
    M_DIESEL_LAPTOPS : UINT := 1103; (* Manufacturer: Diesel Laptops | Location: Irmo, SC USA - 2020-06-10 *)
    M_THE_TORO_COMPANY : UINT := 1104; (* Manufacturer: The Toro Company | Location: Bloomington, MN USA - 2020-06-12 *)
    M_REDEKOP_MANUFACTURING : UINT := 1105; (* Manufacturer: Redekop Manufacturing | Location: Saskatoon, SK Canada - 2020-07-01 *)
    M_GREAT_DANE : UINT := 1106; (* Manufacturer: Great Dane LLC | Location: Chicago, IL USA - 2020-07-01 *)
    M_DR_GER_SAFETY : UINT := 1107; (* Manufacturer: Dräger Safety | Location: Lübeck, Germany - 2020-07-08 *)
    M_ORBCOMM : UINT := 1108; (* Manufacturer: ORBCOMM | Location: Rochelle Park, NJ USA - 2020-07-08 *)
    M_DOCKMATE : UINT := 1109; (* Manufacturer: Dockmate | Location: Boortmeerbeek, Belgium - 2020-07-12 *)
    M_ANALYTIC_SYSTEMS_WARE : UINT := 1110; (* Manufacturer: Analytic Systems Ware (1993) Ltd. | Location: Delta, BC Canada - 2020-07-19 *)
    M_SEPPI_M : UINT := 1111; (* Manufacturer: SEPPI M. | Location: Caldaro, Italy - 2020-07-24 *)
    M_BOLLINGER_MOTORS : UINT := 1112; (* Manufacturer: Bollinger Motors | Location: Oak Park, MI USA - 2020-08-04 *)
    M_IVOLVE_PTY : UINT := 1113; (* Manufacturer: iVolve Pty Ltd | Location: South Brisbane, Australia - 2020-08-04 *)
    M_BOB_S_MACHINE : UINT := 1114; (* Manufacturer: Bob's Machine | Location: Tampa, FL USA - 2020-08-09 *)
    M_GEMS_SENSORS_AND_CONTROLS : UINT := 1115; (* Manufacturer: Gems Sensors & Controls | Location: Plainville, CT USA - 2020-08-14 *)
    M_HR_AGRARTECHNIK : UINT := 1116; (* Manufacturer: HR Agrartechnik GmbH | Location: Velen, Germany - 2020-08-14 *)
    M_LG_CHEM : UINT := 1117; (* Manufacturer: LG Chem, Ltd | Location: Seoul, South Korea - 2020-08-14 *)
    M_L3HARRIS_ASV : UINT := 1118; (* Manufacturer: L3Harris ASV | Location: Portchester, Hampshire UK - 2020-08-18 *)
    M_BALMAR : UINT := 1119; (* Manufacturer: Balmar LLC | Location: Huntsville, AL USA - 2020-08-27 *)
    M_ELETTROMEDIA_S_R_L : UINT := 1120; (* Manufacturer: Elettromedia s.r.l. | Location: Macerata, Italy - 2020-08-27 *)
    M_PLATFORM_SCIENCE : UINT := 1121; (* Manufacturer: Platform Science | Location: La Jolla, CA USA - 2020-09-02 *)
    M_GT : UINT := 1122; (* Manufacturer: GT Inc. | Location: Oak Ridge North, TX USA - 2020-09-02 *)
    M_QP_HYDRAULICS : UINT := 1123; (* Manufacturer: QP Hydraulics | Location: Carol Stream, IL USA - 2020-09-08 *)
    M_FORTRON_AGRICULTURE : UINT := 1124; (* Manufacturer: Fortron Agriculture | Location: Campo Mourão, Brazil - 2020-09-08 *)
    M_GRIFFITH_ELDER_AND : UINT := 1125; (* Manufacturer: Griffith-Elder & Co. Ltd. | Location: Bury St. Edmunds, Suffolk UK - 2020-09-14 *)
    M_AURALIX : UINT := 1126; (* Manufacturer: Auralix | Location: Maribor, Slovenia - 2020-09-14 *)
    M_ELECTROMAAX : UINT := 1127; (* Manufacturer: ElectroMaax | Location: Beamsville, ON Canada - 2020-09-14 *)
    M_CITOON_ELECTRONIC_TECHNOLOGY : UINT := 1128; (* Manufacturer: Citoon Electronic Technology (Tianjin) Co., Ltd. | Location: Tianjin, China - *)
    M_SPECTROLYTIC : UINT := 1129; (* Manufacturer: Spectrolytic GmbH | Location: Wernberg-Koeblitz, Germany - 2020-09-22 *)
    M_VITESCO_TECHNOLOGIES : UINT := 1130; (* Manufacturer: Vitesco Technologies | Location: Regensburg, Germany - 2020-09-22 *)
    M_GULIWER_ELECTRONICS_S_R_O : UINT := 1131; (* Manufacturer: Guliwer electronics s.r.o. | Location: Lanškroun, Czech republic - 2020-09-29 *)
    M_TOKACHI_ZAIDAN : UINT := 1132; (* Manufacturer: Tokachi Zaidan | Location: Obihiro-shi, Japan - 2020-09-29 *)
    M_MEGATRON_ELEKTRONIK_AND : UINT := 1133; (* Manufacturer: MEGATRON Elektronik GmbH & Co. KG | Location: Putzbrunn, Germany - 2020-09-29 *)
    M_MASTER_SCHOOLS_AT_OSTBAHNHOF : UINT := 1134; (* Manufacturer: Master Schools at Ostbahnhof | Location: Munich, Germany - 2020-09-30 *)
    M_JAPAN_AVIATION_ELECTRONICS_INDUSTRY_LIMITED : UINT := 1135; (* Manufacturer: Japan Aviation Electronics Industry, Limited | Location: Tokyo, Japan - 2020-09-30 *)
    M_PRIMOSENSOR : UINT := 1136; (* Manufacturer: Primosensor GmbH | Location: Dieburg, Germany - 2020-10-04 *)
    M_SIKO : UINT := 1137; (* Manufacturer: SIKO GmbH | Location: Buchenbach, Germany - 2020-10-12 *)
    M_MICRO_SENSOR : UINT := 1138; (* Manufacturer: Micro-Sensor GmbH | Location: Hermsdorf, Germany - 2020-10-22 *)
    M_ASP_TECHNOLOGY : UINT := 1139; (* Manufacturer: ASP Technology | Location: Grand Forks, ND USA - 2020-10-14 *)
    M_ACROSS_OCEANS_SYSTEMS : UINT := 1140; (* Manufacturer: Across Oceans Systems Ltd. | Location: North Vancouver, BC Canada - 2020-10-29 *)
    M_MRS_ELECTRONIC_AND : UINT := 1141; (* Manufacturer: MRS Electronic GmbH & Co. KG | Location: Rottweil, Germany - 2020-10-29 *)
    M_TRUMA : UINT := 1142; (* Manufacturer: Truma | Location: Putzbrunn, Germany - 2020-10-29 *)
    M_ELEKTRO_SZOFT_2000 : UINT := 1143; (* Manufacturer: Elektro-Szoft 2000 | Location: Bátmonostor, Hungary - 2020-11-02 *)
    M_TROO : UINT := 1144; (* Manufacturer: Troo Corporation | Location: Ottawa, ON Canada - 2020-11-04 *)
    M_KIWI_YACHTING : UINT := 1145; (* Manufacturer: Kiwi Yachting | Location: Auckland, New Zealand - 2020-11-05 *)
    M_ROMETRON : UINT := 1146; (* Manufacturer: Rometron | Location: Steenderen, the Netherlands - 2020-11-09 *)
    M_DANA : UINT := 1147; (* Manufacturer: Dana Inc. | Location: Maumee, OH USA - 2020-11-10 *)
    M_STERCOM_POWER_SOLUTIONS : UINT := 1148; (* Manufacturer: Stercom Power Solutions GmbH | Location: Weyarn, Germany - 2020-11-10 *)
    M_WUXI_SHENGBANG_ELECTRONICS : UINT := 1149; (* Manufacturer: Wuxi Shengbang Electronics Co., Ltd | Location: Wuxi, China - 2020-11-23 *)
    M_BSB_ARTIFICIAL_INTELLIGENCE : UINT := 1150; (* Manufacturer: BSB Artificial Intelligence GmbH | Location: Linz, Austria - 2020-11-29 *)
    M_ORCA_TECHNOLOGIES : UINT := 1151; (* Manufacturer: Orca Technologies AS | Location: Oslo, Norway - 2020-11-29 *)
    M_VREDO_DODEWAARD_B_V : UINT := 1152; (* Manufacturer: Vredo Dodewaard B.V. | Location: Dodewaard, The Netherlands - 2020-12-18 *)
    M_KAWASAKI_HEAVY_INDUSTRIES : UINT := 1153; (* Manufacturer: Kawasaki Heavy Industries, Ltd. | Location: Kobe, Japan - 2020-12-24 *)
    M_TBS_ELECTRONICS_BV : UINT := 1154; (* Manufacturer: TBS Electronics BV | Location: Zwaag, The Netherlands - 2021-01-05 *)
    M_LACOS : UINT := 1155; (* Manufacturer: LACOS GmbH (formerly LACOS Computerservice GmbH) | Location: Zeulenroda, Germany - *)
    M_NOKIAN_TYRES : UINT := 1156; (* Manufacturer: Nokian Tyres | Location: Nokia, Finland - 2021-01-14 *)
    M_CARRIERGISTICS : UINT := 1157; (* Manufacturer: Carriergistics | Location: Clover, SC USA - 2021-01-22 *)
    M_TECHNOTON_ELECTRONICS : UINT := 1158; (* Manufacturer: Technoton Electronics | Location: Minsk, Belarus - 2021-01-26 *)
    M_BEL_POWER_SOLUTIONS : UINT := 1159; (* Manufacturer: Bel Power Solutions | Location: Dubnica nad Vahom, Slovakia - 2021-02-04 *)
    M_MG_ENERGY_SYSTEMS_B_V : UINT := 1160; (* Manufacturer: MG Energy Systems B.V. | Location: Leeuwarden, The Netherlands - 2021-02-04 *)
    M_GRIESSBACH : UINT := 1161; (* Manufacturer: Griessbach GmbH | Location: Luckenwalde, Germany - 2021-02-08 *)
    M_PEL_TUOTE_OY : UINT := 1162; (* Manufacturer: PEL-tuote Oy | Location: Rantasalmi, Finland - 2021-02-12 *)
    M_DFX_TECHNOLOGIES : UINT := 1163; (* Manufacturer: DFX Technologies LLC | Location: Roswell, GA USA - 2021-02-18 *)
    M_SEG_AUTOMOTIVE : UINT := 1164; (* Manufacturer: SEG Automotive | Location: Stuttgart, Germany - 2021-03-08 *)
    M_INNOTOTAL : UINT := 1165; (* Manufacturer: InnoTotal AB | Location: Kungälv, Sweden - 2021-03-14 *)
    M_WACHENDORFF_AUTOMATION_AND : UINT := 1166; (* Manufacturer: Wachendorff Automation GmbH & Co. KG | Location: Geisenheim, Germany - 2021-03-16 *)
    M_TEVVA_MOTORS : UINT := 1167; (* Manufacturer: Tevva Motors | Location: Chelmsford, Essex UK - 2021-03-19 *)
    M_MASATS : UINT := 1168; (* Manufacturer: Masats S.A. | Location: Sant Salvador de Guardiola, Barcelona Spain - 2021-03-23 *)
    M_SEA_MACHINE_ROBOTICS : UINT := 1169; (* Manufacturer: Sea Machine Robotics Inc. | Location: Boston, MA USA - 2021-04-01 *)
    M_POSEIDON_OCEAN_SYSTEMS : UINT := 1170; (* Manufacturer: Poseidon Ocean Systems Ltd. | Location: Campbell River, BC Canada - 2021-04-08 *)
    M_VISTA_MANUFACTURING : UINT := 1171; (* Manufacturer: Vista Manufacturing | Location: Elkhart, IN USA - 2021-04-13 *)
    M_HYZON_MOTORS : UINT := 1172; (* Manufacturer: Hyzon Motors | Location: Honeoye Falls, NY USA - 2021-04-13 *)
    M_PHILIPPI_ELEKTRISCHE_SYSTEME : UINT := 1173; (* Manufacturer: philippi elektrische systeme gmbh | Location: Remseck am Neckar, Germany - *)
    M_AGRICON : UINT := 1174; (* Manufacturer: Agricon GmbH | Location: Ostrau, Germany - 2021-04-19 *)
    M_MAGTEC_PRODUCTS : UINT := 1175; (* Manufacturer: MAGTEC Products, Inc. | Location: Calgary, AB Canada - 2021-04-20 *)
    M_ASUNS : UINT := 1176; (* Manufacturer: Asuns Corp. | Location: Dundee, IL USA - 2021-05-02 *)
    M_RNG_INTERNATIONAL : UINT := 1177; (* Manufacturer: RNG International Inc. | Location: Ontario, CA USA - 2021-05-02 *)
    M_ERO : UINT := 1178; (* Manufacturer: ERO GmbH | Location: Simmern, Germany - 2021-05-02 *)
    M_QS_CONTROL_SRL : UINT := 1179; (* Manufacturer: QS Control srl | Location: Narni, Italy - 2021-05-04 *)
    M_MURATA_POWER_SOLUTIONS : UINT := 1180; (* Manufacturer: Murata Power Solutions Inc. | Location: Westborough, MA USA - 2021-05-25 *)
    M_BANJO : UINT := 1181; (* Manufacturer: Banjo Corporation | Location: Crawfordsville, IN USA - 2021-05-25 *)
    M_ROTTMANN_AUTOMATION : UINT := 1182; (* Manufacturer: Rottmann Automation | Location: Ochtrup, Germany - 2021-05-27 *)
    M_ZIPWAKE : UINT := 1183; (* Manufacturer: Zipwake AB | Location: Gothenburg, Sweden - 2021-06-07 *)
    M_AMA : UINT := 1184; (* Manufacturer: AMA S.p.A. | Location: Campogalliano, Italy - 2021-06-07 *)
    M_WFCO_ELECTRONICS : UINT := 1185; (* Manufacturer: WFCO Electronics | Location: Tang Xia Town, China - 2021-06-07 *)
    M_SAILMON_BV : UINT := 1186; (* Manufacturer: Sailmon BV | Location: Den Haag, The Netherlands - 2021-06-15 *)
    M_TITAN_PROJECT : UINT := 1187; (* Manufacturer: TiTAN-Project LLC | Location: Moscow, Russian Federation - 2021-07-10 *)
    M_G_SNS : UINT := 1188; (* Manufacturer: G-SNS | Location: Munich, Germany - 2021-07-20 *)
    M_AUTOTRASPORTI_CAVALLO_G_AND_V : UINT := 1189; (* Manufacturer: Autotrasporti Cavallo G&V | Location: Boves (CN), Italy - 2021-07-26 *)
    M_SIRROS_IOT : UINT := 1190; (* Manufacturer: Sirros IoT | Location: Novo Hamburgo, Brazil - 2021-07-26 *)
    M_PACOMA_USA : UINT := 1191; (* Manufacturer: Pacoma USA, Inc. | Location: Halifax, PA USA - 2021-08-03 *)
    M_AIRMONIQ_PRO_KFT : UINT := 1192; (* Manufacturer: Airmoniq Pro Kft. | Location: Pécs, Hungary - 2021-08-12 *)
    M_EMOTAS_EMBEDDED_COMMUNICATION : UINT := 1193; (* Manufacturer: emotas embedded communication GmbH | Location: Merseburg, Germany - 2021-08-26 *)
    M_SIERRA_MARINE : UINT := 1194; (* Manufacturer: Sierra Marine | Location: Litchfield, IL - 2021-08-26 *)
    M_D_VELSDORF : UINT := 1195; (* Manufacturer: düvelsdorf | Location: Ottersberg, Germany - 2021-09-10 *)
    M_TERRA_CARE : UINT := 1196; (* Manufacturer: Terra Care GmbH | Location: Neukirchen, Austria - 2021-09-10 *)
    M_SOLGE : UINT := 1197; (* Manufacturer: SOLGE Corporation | Location: Daegu, South Korea - 2021-09-10 *)
    M_COMLINK_EQUIPAMENTOS_ELETR_NICOS_LTDA : UINT := 1198; (* Manufacturer: ComLink Equipamentos Eletrônicos Ltda | Location: Caxias do Sul, Brazil - *)
    M_ELEO_TECHNOLOGIES_B_V : UINT := 1199; (* Manufacturer: ELEO Technologies B.V. | Location: Helmond, The Netherlands - 2021-09-10 *)
    M_XINUO_INFORMATION_TECHNOLOGY_LIMITED : UINT := 1200; (* Manufacturer: Xinuo Information Technology (Xiamen) Corporation Limited | Location: Xiamen, China *)
    M_EMISENSE_TECHNOLOGIES : UINT := 1201; (* Manufacturer: Emisense Technologies, LLC | Location: Ladera Ranch, CA USA - 2021-09-30 *)
    M_OSCAR_ELECTRONICS_SRL : UINT := 1202; (* Manufacturer: OSCAR ELECTRONICS SRL (formerly OSCAR Elettronica) | Location: Carpenedolo, Italy - *)
    M_EQUIPMENT_TECHNOLOGIES : UINT := 1203; (* Manufacturer: Equipment Technologies, Inc. | Location: Mooresville, IN USA - 2021-09-30 *)
    M_MILLER_TECHNOLOGY_INCORPORATED : UINT := 1204; (* Manufacturer: Miller Technology Incorporated | Location: North Bay, ON Canada - 2021-09-30 *)
    M_CARBON_AUTONOMOUS_ROBOTIC_SYSTEMS : UINT := 1205; (* Manufacturer: Carbon Autonomous Robotic Systems | Location: Seattle, WA USA - 2021-09-30 *)
    M_STE_SOLUTIONS_B_V : UINT := 1206; (* Manufacturer: STE Solutions B.V. | Location: Wehl, The Netherlands - 2021-09-30 *)
    M_UEC_ELECTRONICS : UINT := 1207; (* Manufacturer: UEC Electronics | Location: Hanahan, SC USA - 2021-09-30 *)
    M_AFFLIELD_KFT : UINT := 1208; (* Manufacturer: Afflield Kft. (MachineryGuide) | Location: Budapest, Hungary - 2021-09-30 *)
    M_BAUSER_AND : UINT := 1209; (* Manufacturer: Bauser GmbH & Co. KG | Location: Empfingen, Germany - 2021-09-30 *)
    M_AMBRA_SOLUTIONS : UINT := 1210; (* Manufacturer: Ambra Solutions | Location: Trois-Rivieres, QC Canada - 2021-10-13 *)
    M_KIWON_ELECTRONICS : UINT := 1211; (* Manufacturer: Kiwon Electronics Co., Ltd. | Location: Iksan, Republic of Korea - 2021-10-13 *)
    M_TAO_PERFORMANCE_LIMITED : UINT := 1212; (* Manufacturer: TAO Performance Limited | Location: Paihia, New Zealand - 2021-10-26 *)
    M_APOLLO_TYRES : UINT := 1213; (* Manufacturer: Apollo Tyres Ltd | Location: Gurgaon, India - 2021-10-26 *)
    M_ELEMENT_1 : UINT := 1214; (* Manufacturer: Element 1 | Location: Bend, OR USA - 2021-10-31 *)
    M_POWER_CONTROL_SYSTEMS : UINT := 1215; (* Manufacturer: Power Control Systems | Location: San Vendemiano, Italy - 2021-11-06 *)
    M_SMP_POLAND_SP_Z_O_O : UINT := 1216; (* Manufacturer: SMP Poland sp. z o.o. | Location: Warsaw, Poland - 2021-11-21 *)
    M_FSG_FERNSTEUERGER_TE_KURT_OELSCH : UINT := 1217; (* Manufacturer: FSG Fernsteuergeräte Kurt Oelsch GmbH | Location: Berlin, Germany - 2021-11-24 *)
    M_SEPTENTRIO : UINT := 1218; (* Manufacturer: Septentrio | Location: Leuven, Belgium - 2021-11-28 *)
    M_WEIDMUELLER_INTERFACE_AND : UINT := 1219; (* Manufacturer: Weidmueller Interface GmbH & Co. KG | Location: Detmold, Germany - 2021-11-30 *)
    M_CATAMARAN_ELECTRONICS : UINT := 1220; (* Manufacturer: Catamaran Electronics LLC | Location: West Melbourne, FL USA - 2021-12-03 *)
    M_NORCOLD : UINT := 1221; (* Manufacturer: Norcold Inc. | Location: Sidney, OH USA - 2021-12-03 *)
    M_TOUGH_TECH : UINT := 1222; (* Manufacturer: Tough Tech Ltd. | Location: Whitchurch, Shropshire UK - 2021-12-03 *)
    M_TOYO_AGRICULTURAL_MACHINERY_MANUFACTURING : UINT := 1223; (* Manufacturer: Toyo Agricultural Machinery Manufacturing Co., Ltd. | Location: Obihiro, Japan - *)
    M_NEUSER_ELEKTROTECHNIK : UINT := 1224; (* Manufacturer: Neuser Elektrotechnik GmbH | Location: Birkenbeul, Germany - 2021-12-03 *)
    M_SEEDMASTER_MANUFACTURING : UINT := 1225; (* Manufacturer: SeedMaster Manufacturing Ltd. | Location: Emerald Park, SK Canada - 2021-12-09 *)
    M_PIIPPO_HYDRAULIC : UINT := 1226; (* Manufacturer: Piippo Hydraulic | Location: Kiuruvesi, Finland - 2021-12-09 *)
    M_YAHATA : UINT := 1227; (* Manufacturer: YAHATA Co., Ltd. | Location: YaoCity, Osaka Japan - 2021-12-09 *)
    M_INTILION : UINT := 1228; (* Manufacturer: INTILION GmbH | Location: Zwickau, Germany - 2021-12-13 *)
    M_ARCON_DESIGNS : UINT := 1229; (* Manufacturer: Arcon Designs, LLC | Location: Bloomington, IN USA - 2021-12-23 *)
    M_NICK_ABBEY_DIGITAL_AGRICULTURE : UINT := 1230; (* Manufacturer: Nick Abbey Digital Agriculture Ltd | Location: Scarborough, Yorkshire UK - *)
    M_EXCIDOR : UINT := 1231; (* Manufacturer: Excidor AB | Location: Bollnäs, Sweden - 2021-12-23 *)
    M_TREFFLER_MASCHINENBAU_AND : UINT := 1232; (* Manufacturer: Treffler Maschinenbau GmbH & Co. KG | Location: Pöttmes-Echsheim, Germany - *)
    M_NKE_MARINE_ELECTRONICS : UINT := 1233; (* Manufacturer: nke Marine Electronics | Location: Hennebont, France - 2021-12-29 *)
    M_AMERICAN_BATTERY_SOLUTIONS : UINT := 1234; (* Manufacturer: American Battery Solutions | Location: Lake Orion, MI USA - 2022-01-09 *)
    M_NESAN_AUTOMOTIVE : UINT := 1235; (* Manufacturer: NESAN Automotive Inc. | Location: Izmir, Turkey - 2022-01-17 *)
    M_AGROSYSTEM : UINT := 1236; (* Manufacturer: Agrosystem | Location: Ribeirao Preto, Brazil - 2022-01-17 *)
    M_CHANGZHOU_LAMBDA_ELECTRONIC : UINT := 1237; (* Manufacturer: Changzhou Lambda Electronic Co., Ltd | Location: Changzhou, China - 2022-01-17 *)
    M_HONDA_ELECTRONICS : UINT := 1238; (* Manufacturer: Honda Electronics Co., Ltd | Location: Toyohashi, Aichi Japan - 2022-01-21 *)
    M_SUPERTRACK_APS : UINT := 1239; (* Manufacturer: SuperTrack Aps | Location: Egaa, Denmark - 2022-01-21 *)
    M_TIMOTION : UINT := 1240; (* Manufacturer: TiMOTION | Location: New Taipei City, Taiwan - 2022-01-21 *)
    M_INEO_SYSTRANS : UINT := 1241; (* Manufacturer: Ineo Systrans | Location: Achères, France - 2022-01-28 *)
    M_SUPER_START_BATTERIES : UINT := 1242; (* Manufacturer: Super Start Batteries | Location: Lansvale, NSW Australia - 2022-01-28 *)
    M_AVMAP_S_R_L : UINT := 1243; (* Manufacturer: AvMap S.r.l. | Location: Carrara (MS), Italy - 2022-01-28 *)
    M_PLANTI_CENTER : UINT := 1244; (* Manufacturer: Planti Center | Location: Marialva, Brazil - 2022-02-06 *)
    M_RARITAN_ENGINEERING_COMPANY : UINT := 1245; (* Manufacturer: Raritan Engineering Company, Inc | Location: Millville, NJ USA - 2022-02-14 *)
    M_ROTHER_INDUSTRIES_AND_TECHNOLOGY : UINT := 1246; (* Manufacturer: Rother Industries & Technology | Location: Cordoba, Spain - 2022-02-14 *)
    M_GRIFA : UINT := 1247; (* Manufacturer: GRIFA | Location: Pfullendorf, Germany - 2022-02-14 *)
    M_O_M_F_B_HYDRAULIC_COMPONENTS : UINT := 1248; (* Manufacturer: O.M.F.B. S.p.A. Hydraulic Components | Location: Provaglio d'Iseo (BS), Italy - *)
    M_INTEGRATED_POWER_SOLUTIONS_AG : UINT := 1249; (* Manufacturer: Integrated Power Solutions AG | Location: Port, Switzerland - 2022-03-06 *)
    M_ELHO : UINT := 1250; (* Manufacturer: ELHO | Location: Pännäinen, Finland - 2022-03-29 *)
    M_VALMET_AUTOMOTIVE_EV_POWER : UINT := 1251; (* Manufacturer: Valmet Automotive EV Power Ltd | Location: Uusikaupunki, Finland - 2022-04-11 *)
    M_APV_TECHNISCHE_PRODUKTE : UINT := 1252; (* Manufacturer: APV - Technische Produkte GmbH | Location: Hötzelsdorf, Austria - 2022-04-11 *)
    M_TRAFAG_AG : UINT := 1253; (* Manufacturer: Trafag AG | Location: Bubikon, Switzerland - 2022-04-11 *)
    M_ARADEX_AG : UINT := 1254; (* Manufacturer: ARADEX AG | Location: Lorch, Germany - 2022-04-11 *)
    M_ALTEC_INDUSTRIES : UINT := 1255; (* Manufacturer: Altec Industries, Inc. | Location: Birmingham, AL USA - 2022-04-12 *)
    M_DIMENSIONS_AGRI_TECHNOLOGIES : UINT := 1256; (* Manufacturer: Dimensions Agri Technologies AS | Location: Oslo, Norway - 2022-04-12 *)
    M_KOSTAL : UINT := 1257; (* Manufacturer: KOSTAL | Location: Hagen, Germany - 2022-04-12 *)
    M_AGC_TECHNOLOGIES : UINT := 1258; (* Manufacturer: AGC Technologies | Location: Madrid, Spain - 2022-04-12 *)
    M_GRAYSON_AUTOMOTIVE_SERVICES_LIMITED : UINT := 1259; (* Manufacturer: Grayson Automotive Services Limited | Location: Birmingham, West Midlands UK - *)
    M_INTERACTIVE_TECHNOLOGIES : UINT := 1260; (* Manufacturer: Interactive Technologies, Inc. | Location: Olathe, KS USA - 2022-04-12 *)
    M_AGXEED : UINT := 1261; (* Manufacturer: AgXeed | Location: Grubbenvorst, The Netherlands - 2026-02-09 *)
    M_FORT_ROBOTICS : UINT := 1262; (* Manufacturer: Fort Robotics | Location: Philadelphia, PA USA - 2022-04-15 *)
    M_BOS_BALANCE_OF_STORAGE_SYSTEMS_AG : UINT := 1263; (* Manufacturer: BOS Balance of Storage Systems AG | Location: Neu-Ulm, Germany - 2022-04-25 *)
    M_MICROELECT : UINT := 1264; (* Manufacturer: Microelect | Location: Villa Gobernador Gálvez, Argentina - 2022-04-25 *)
    M_IPETRONIK_AND : UINT := 1265; (* Manufacturer: IPETRONIK GmbH & Co KG | Location: Baden-Baden, Germany - 2022-05-02 *)
    M_HYUNDAI_DOOSAN_INFRACORE : UINT := 1266; (* Manufacturer: Hyundai Doosan Infracore | Location: Incheon, Republic of Korea - 2022-05-02 *)
    M_WACKER_NEUSON_SE : UINT := 1267; (* Manufacturer: Wacker Neuson SE | Location: Munich, Germany - 2022-05-02 *)
    M_BACK_40_PRECISION : UINT := 1268; (* Manufacturer: Back 40 Precision Inc. | Location: Baldwin, IL USA - 2022-05-04 *)
    M_VIS_HYDRAULICS_S_R_L : UINT := 1269; (* Manufacturer: VIS Hydraulics s.r.l. | Location: Pavullo Nel Frignano, Italy - 2022-05-09 *)
    M_VERSALIFT_DENMARK : UINT := 1270; (* Manufacturer: Versalift Denmark A/S | Location: Farsø, Denmark - 2022-05-09 *)
    M_RAVEN_CONNECTED : UINT := 1271; (* Manufacturer: Raven Connected | Location: Ottawa, ON Canada - 2022-05-14 *)
    M_SAMSARA : UINT := 1272; (* Manufacturer: Samsara Inc. | Location: San Francisco, CA USA - 2022-05-17 *)
    M_CLEARFLAME_ENGINES : UINT := 1273; (* Manufacturer: Clearflame Engines Inc | Location: Geneva, IL USA - 2022-05-22 *)
    M_LDL_TECHNOLOGY : UINT := 1274; (* Manufacturer: LDL Technology | Location: Ramonville-Saint-Agne, France - 2022-05-22 *)
    M_O_M_P_OFFICINE_MAZZOCCO_PAGNONI_S_R_L : UINT := 1275; (* Manufacturer: O.M.P. Officine Mazzocco Pagnoni S.r.l. | Location: Funo, Italy - 2022-05-22 *)
    M_ASPIN_KEMP_AND_ASSOCIATES : UINT := 1276; (* Manufacturer: Aspin Kemp & Associates | Location: Montague, PE Canada - 2022-06-10 *)
    M_BMZ_GERMANY : UINT := 1277; (* Manufacturer: BMZ Germany GmbH | Location: Karlstein am Main, Germany - 2022-06-10 *)
    M_COMROD_COMMUNICATION_GROUP : UINT := 1278; (* Manufacturer: Comrod Communication Group | Location: Stavanger, Norway - 2022-06-21 *)
    M_OGNIBENE_POWER : UINT := 1279; (* Manufacturer: Ognibene Power S.p.A. | Location: Reggio Emilia (RE), Italy - 2022-06-21 *)
    M_SANTEST : UINT := 1280; (* Manufacturer: SANTEST CO., LTD. | Location: Osaka-shi, Osaka Japan - 2022-07-05 *)
    M_IQUUS : UINT := 1281; (* Manufacturer: iQuus | Location: Neerijnen, The Netherlands - 2022-07-05 *)
    M_COTEK_ELECTRONIC_IND : UINT := 1282; (* Manufacturer: COTEK ELECTRONIC IND. CO., LTD | Location: Taoyuan City, Taiwan - 2022-07-07 *)
    M_LTG_TECH : UINT := 1283; (* Manufacturer: LTG Tech | Location: Metz, France - 2022-07-18 *)
    M_ROBOT_MAKERS : UINT := 1284; (* Manufacturer: Robot Makers GmbH | Location: Kaiserslautern, Germany - 2022-07-18 *)
    M_GRACO : UINT := 1285; (* Manufacturer: Graco Inc. | Location: Minnepolis, MN USA - 2022-07-18 *)
    M_NEXAT : UINT := 1286; (* Manufacturer: NEXAT GmbH | Location: Rieste, Germany - 2022-07-21 *)
    M_SPARTAN_RADAR : UINT := 1287; (* Manufacturer: Spartan Radar | Location: Los Alamitos, CA USA - 2022-08-03 *)
    M_ANELLO_PHOTONICS : UINT := 1288; (* Manufacturer: ANELLO Photonics | Location: Santa Clara, CA USA - 2022-08-03 *)
    M_LOADRITE : UINT := 1289; (* Manufacturer: Loadrite (Auckland) Ltd. | Location: Auckland, New Zealand - 2022-08-03 *)
    M_WAVETAMER_PARTNERS : UINT := 1290; (* Manufacturer: WaveTamer Partners LLC | Location: Greensboro, NC USA - 2022-08-03 *)
    M_FORWARD_THINKING_SYSTEMS : UINT := 1291; (* Manufacturer: Forward Thinking Systems LLC | Location: Jericho, NY USA - 2022-08-08 *)
    M_SUMITOMO_CONSTRUCTION_MACHINERY : UINT := 1292; (* Manufacturer: SUMITOMO CONSTRUCTION MACHINERY Co., Ltd. | Location: Tokyo, Japan - 2022-08-09 *)
    M_POSITAL : UINT := 1293; (* Manufacturer: POSITAL | Location: Aachen, Germany - 2022-08-18 *)
    M_TR_ELECTRONIC : UINT := 1294; (* Manufacturer: TR-Electronic GmbH | Location: Trossingen, Germany - 2022-09-01 *)
    M_SIP_D_D : UINT := 1295; (* Manufacturer: SIP d.d. | Location: Šempeter v Savinjski Dolini, Slovenia - 2022-09-01 *)
    M_HEXAGON : UINT := 1296; (* Manufacturer: Hexagon | Location: Florianópolis, Brazil - 2022-09-14 *)
    M_MICRO_EPSILON_MESSTECHNIK_AND : UINT := 1297; (* Manufacturer: Micro-Epsilon Messtechnik GmbH & Co. KG | Location: Ortenburg, Germany - 2022-09-14 *)
    M_SFOGGIA_AGRICULTURE_DIVISION_S_R_L : UINT := 1298; (* Manufacturer: SFOGGIA Agriculture Division S.r.l. | Location: Montebelluna, Italy - 2022-09-14 *)
    M_ENERGY_SOLUTIONS : UINT := 1299; (* Manufacturer: Energy Solutions | Location: Rochester, Kent UK - 2022-09-15 *)
    M_WATT_FUEL_CELL : UINT := 1300; (* Manufacturer: Watt Fuel Cell Corporation | Location: Mount Pleasant, PA USA - 2022-09-15 *)
    M_TECUMSEH_DO_BRASIL_LTDA : UINT := 1301; (* Manufacturer: Tecumseh do Brasil Ltda | Location: São Carlos, São Paulo Brazil - 2022-09-23 *)
    M_PROMARINER : UINT := 1302; (* Manufacturer: ProMariner | Location: Auburn, NH USA - 2022-09-23 *)
    M_CARBON_BEE_AGTECH : UINT := 1303; (* Manufacturer: Carbon Bee AgTech | Location: Valence, France - 2022-10-19 *)
    M_PALFINGER_EUROPE : UINT := 1304; (* Manufacturer: Palfinger Europe GmbH | Location: Salzburg, Austria - 2022-10-19 *)
    M_DRAGONFLY_ENERGY_1305 : UINT := 1305; (* Manufacturer: dragonfly Energy | Location: Reno, NV USA - 2022-10-22 *)
    M_KODEN_ELECTRONICS : UINT := 1306; (* Manufacturer: Koden Electronics Co., Ltd. | Location: Tokyo, Japan - 2022-10-22 *)
    M_SMART_AG_SYSTEMS : UINT := 1307; (* Manufacturer: Smart AG Systems | Location: Yeerongpilly, QLD Australia - 2022-10-31 *)
    M_AGTECNIC : UINT := 1308; (* Manufacturer: Agtecnic | Location: Brisbane, QLD Australia - 2022-11-04 *)
    M_SHANGHAI_ZHICHUAN_ELECTRONIC_TECH : UINT := 1309; (* Manufacturer: Shanghai Zhichuan Electronic Tech Co., Ltd. | Location: Shanghai, China - *)
    M_LPL_SYSTEMS : UINT := 1310; (* Manufacturer: LPL Systems (formerly Loughborough Projects Ltd) | Location: Loughborough, *)
    M_HUMPHREE : UINT := 1311; (* Manufacturer: Humphree AB | Location: Gothenburg, Sweden - 2022-11-22 *)
    M_CONTROL_DEVICES_PTY : UINT := 1312; (* Manufacturer: Control Devices Pty Ltd | Location: Alexandria, NSW Australia - 2022-12-01 *)
    M_UNITED_STATES_ARMY_GROUND_VEHICLE_SYSTEMS_CENTER : UINT := 1313; (* Manufacturer: United States Army - Ground Vehicle Systems Center | Location: Warren, MI USA - *)
    M_NEWTON_CROUCH_COMPANY : UINT := 1314; (* Manufacturer: Newton Crouch Company, LLC | Location: Griffin, GA USA - 2022-12-07 *)
    M_SMPC_TECHNOLOGIES : UINT := 1315; (* Manufacturer: SMPC Technologies Ltd. | Location: Burnaby, BC Canada - 2022-12-07 *)
    M_HINKLEY_YACHTS : UINT := 1316; (* Manufacturer: Hinkley Yachts | Location: Portsmouth, RI USA - 2022-12-07 *)
    M_GMM_GLOBAL_MARITIME_MANAGEMENT : UINT := 1317; (* Manufacturer: GMM - Global Maritime Management GmbH | Location: Trittau, Germany - 2022-12-07 *)
    M_ATLIS_MOTOR_VEHICLES : UINT := 1318; (* Manufacturer: Atlis Motor Vehicles | Location: Mesa, AZ USA - 2022-12-12 *)
    M_I_O_CONTROLS : UINT := 1319; (* Manufacturer: I/O Controls Corporation | Location: Azusa, CA USA - 2022-12-12 *)
    M_TRISKEL_MARINE : UINT := 1320; (* Manufacturer: Triskel Marine Ltd | Location: Hayle, Cornwall UK - 2022-12-19 *)
    M_PATLITE : UINT := 1321; (* Manufacturer: PATLITE Corporation | Location: Osaka, Japan - 2022-12-19 *)
    M_MOVIMATICA : UINT := 1322; (* Manufacturer: Movimatica | Location: Cuneo, Italy - 2023-01-03 *)
    M_BRITER_PRODUCTS : UINT := 1323; (* Manufacturer: Briter Products, Inc. | Location: South Bend, IN USA - 2023-01-03 *)
    M_BOURGAULT_INDUSTRIES : UINT := 1324; (* Manufacturer: Bourgault Industries | Location: Saint Brieux, SK Canada - 2023-01-14 *)
    M_OPW : UINT := 1325; (* Manufacturer: OPW (formerly BASE Engineering Inc.) | Location: Hamilton, OH USA - 2025-04-09 *)
    M_HBC_RADIOMATIC : UINT := 1326; (* Manufacturer: HBC-radiomatic GmbH | Location: Crailsheim, Germany - 2023-01-14 *)
    M_FRANS_VERVAET_B_V : UINT := 1327; (* Manufacturer: Frans Vervaet B.V. | Location: Biervliet, The Netherlands - 2023-01-20 *)
    M_PERPLANT_APS : UINT := 1328; (* Manufacturer: PerPlant ApS | Location: København K, Denmark - 2023-01-20 *)
    M_IDM_S_R_L : UINT := 1329; (* Manufacturer: IDM S.r.l. | Location: Montebelluna, Italy - 2023-01-20 *)
    M_WARWICK_CONTROL_TECHNOLOGIES : UINT := 1330; (* Manufacturer: Warwick Control Technologies | Location: Halesowen, West Midlands UK - 2023-01-20 *)
    M_DOLPHIN_CHARGER : UINT := 1331; (* Manufacturer: Dolphin Charger | Location: Annecy, France - 2023-01-20 *)
    M_FAIRBANKS_SCALES : UINT := 1332; (* Manufacturer: Fairbanks Scales, Inc. | Location: Overland Park, KS USA - 2023-01-26 *)
    M_XFARM_TECHNOLOGIES : UINT := 1333; (* Manufacturer: xFarm Technologies SA | Location: Manno, Switzerland - 2023-02-17 *)
    M_GREER_COMPANY : UINT := 1334; (* Manufacturer: Greer Company | Location: Jenks, OK USA - 2023-01-27 *)
    M_CPDEVICE : UINT := 1335; (* Manufacturer: CPDEVICE | Location: Beijing, China - 2023-02-03 *)
    M_AEGIS_POWER_SYSTEMS : UINT := 1336; (* Manufacturer: Aegis Power Systems, Inc. | Location: Murphy, NC USA - 2023-02-03 *)
    M_BARNACLE_SYSTEMS : UINT := 1337; (* Manufacturer: Barnacle Systems Inc. | Location: Victoria, BC Canada - 2023-02-22 *)
    M_VOLTA_TRUCKS : UINT := 1338; (* Manufacturer: Volta Trucks AB | Location: Stockholm, Sweden - 2023-02-24 *)
    M_TILLETT_AND_HAGUE_TECHNOLOGY_LIMITED : UINT := 1339; (* Manufacturer: Tillett and Hague Technology Limited | Location: Bedford, Bedfordshire UK - *)
    M_ORELTEK_ELEKTRONIK_VE_YAZILIM_TEKNOLOJILERI : UINT := 1340; (* Manufacturer: ORELTEK Elektronik ve Yazılım Teknolojileri | Location: Serdivan, Turkey - *)
    M_AG_EXPRESS_ELECTRONICS : UINT := 1341; (* Manufacturer: Ag Express Electronics | Location: Des Moines, IA USA - 2023-03-04 *)
    M_DKE_DATA_AND : UINT := 1342; (* Manufacturer: DKE-Data GmbH & Co. KG | Location: Osnabrück, Germany - 2023-03-04 *)
    M_HEAVY_DATA : UINT := 1343; (* Manufacturer: Heavy Data GmbH | Location: Oberursel, Germany - 2023-03-04 *)
    M_HAULOTTE_GROUP : UINT := 1344; (* Manufacturer: Haulotte Group | Location: Lorette, France - 2023-03-07 *)
    M_PRIGNITZ_MIKROSYSTEMTECHNIK : UINT := 1345; (* Manufacturer: PRIGNITZ Mikrosystemtechnik GmbH | Location: Wittenberge, Germany - 2023-03-16 *)
    M_EINBOECK : UINT := 1346; (* Manufacturer: Einboeck GmbH | Location: Dorf an der Pram, Austria - 2023-03-16 *)
    M_MUNCKHOF_FRUIT_TECH_INNOVATORS : UINT := 1347; (* Manufacturer: Munckhof Fruit Tech Innovators | Location: Horst, The Netherlands - 2023-03-16 *)
    M_RADIAN_IOT : UINT := 1348; (* Manufacturer: Radian IoT, Inc. | Location: Okauche, WI USA - 2023-03-16 *)
    M_ANNABURGER_NUTZFAHRZEUG : UINT := 1349; (* Manufacturer: ANNABURGER Nutzfahrzeug GmbH | Location: Annaburg, Germany - 2023-03-21 *)
    M_AGRONETIC : UINT := 1350; (* Manufacturer: AGRONETIC | Location: Liege, Belgium - 2023-03-21 *)
    M_MOTORENFABRIK_HATZ_AND : UINT := 1351; (* Manufacturer: Motorenfabrik Hatz GmbH & Co. KG | Location: Ruhstorf, Germany - 2023-03-29 *)
    M_NISHIYAMA : UINT := 1352; (* Manufacturer: NISHIYAMA Corporation | Location: Tokyo, Japan - 2023-03-29 *)
    M_OCEAN_LED_MARINE : UINT := 1353; (* Manufacturer: Ocean LED Marine Ltd | Location: Hinkley, Leicestershire UK - 2023-04-09 *)
    M_T_CNICAS_DE_ELECTR_NICA_Y_AUTOMATISMOS : UINT := 1354; (* Manufacturer: Técnicas de Electrónica y Automatismos, S.A. | Location: Barcelona, Spain - *)
    M_DROP_AGRICULTURA_LTDA : UINT := 1355; (* Manufacturer: DROP Agricultura Ltda | Location: Piracicaba, Brazil - 2023-04-22 *)
    M_NORDIC_LIGHTS : UINT := 1356; (* Manufacturer: Nordic Lights Ltd | Location: Jakobstad, Finland - 2023-04-22 *)
    M_TIRECHECK : UINT := 1357; (* Manufacturer: TireCheck | Location: Heidenheim, Germany - 2023-05-07 *)
    M_FONTAINE_FIFTH_WHEEL : UINT := 1358; (* Manufacturer: Fontaine Fifth Wheel | Location: Jasper, AL USA - 2023-05-07 *)
    M_BLUENAV : UINT := 1359; (* Manufacturer: BlueNav | Location: Arcachon, France - 2023-05-07 *)
    M_LEMCA_VISION : UINT := 1360; (* Manufacturer: Lemca Vision | Location: Glabais, Belgium - 2023-05-07 *)
    M_NANTONG_SAIYANG_ELECTRONICS : UINT := 1361; (* Manufacturer: Nantong Saiyang Electronics Co., Ltd. | Location: Nantong, China - 2023-05-18 *)
    M_ZPARQ : UINT := 1362; (* Manufacturer: Zparq AB | Location: Stockholm, Sweden - 2023-05-18 *)
    M_CALIX : UINT := 1363; (* Manufacturer: Calix AB | Location: Eskilstuna, Sweden - 2023-05-18 *)
    M_YASHU_SYSTEMS : UINT := 1364; (* Manufacturer: Yashu Systems | Location: Archbald, PA USA - 2023-06-02 *)
    M_JVCKENWOOD : UINT := 1365; (* Manufacturer: JVCKENWOOD Corporation | Location: Kanagawa, Japan - 2023-06-02 *)
    M_TELEMECANIQUE_SENSORS_AND_SWITCHES : UINT := 1366; (* Manufacturer: Telemecanique Sensors & Switches | Location: Rueil-Malmaison, France - 2023-06-16 *)
    M_DEWULF_NV : UINT := 1367; (* Manufacturer: Dewulf NV | Location: Roeselare, Belgium - 2023-06-25 *)
    M_RAD_PROPULSION : UINT := 1368; (* Manufacturer: RAD Propulsion Ltd | Location: Sarisbury Green, Southampton UK - 2023-06-25 *)
    M_ELECTRIC_YACHT : UINT := 1369; (* Manufacturer: Electric Yacht | Location: Golden Valley, MN USA - 2023-06-25 *)
    M_EMTECH : UINT := 1370; (* Manufacturer: Emtech S.A. | Location: Bahia Blanca, Buenos Aires Argentina - 2023-08-04 *)
    M_FIRST_MODE : UINT := 1371; (* Manufacturer: First Mode | Location: Seattle, WA USA - 2023-06-25 *)
    M_ELCO_MOTOR_YACHTS : UINT := 1372; (* Manufacturer: Elco Motor Yachts | Location: Shelton, CT USA - 2023-06-30 *)
    M_CENTEK_INDUSTRIES : UINT := 1373; (* Manufacturer: Centek Industries | Location: Thomasville, GA USA - 2023-07-06 *)
    M_CASAPPA : UINT := 1374; (* Manufacturer: CASAPPA S.p.A. | Location: Parma, Italy - 2023-07-06 *)
    M_KODA_ELECTRIC_A_S_1375 : UINT := 1375; (* Manufacturer: ŠKODA ELECTRIC a.s. | Location: Plzeň, Czech republic - 2023-08-14 *)
    M_SUNS_INTERNATIONAL : UINT := 1376; (* Manufacturer: SUNS International, LLC | Location: Chelmsford, MA USA - 2023-07-06 *)
    M_ABD_SOLUTIONS : UINT := 1377; (* Manufacturer: ABD Solutions | Location: Bradford on Avon, Wiltshire UK - 2023-07-24 *)
    M_BERTINI : UINT := 1378; (* Manufacturer: Bertini SA | Location: Rosario, Santa Fe Argentina - 2023-07-24 *)
    M_NOVAG_SAS : UINT := 1379; (* Manufacturer: Novag SAS | Location: Fressines, France - 2023-07-24 *)
    M_ADVES_AND : UINT := 1380; (* Manufacturer: ADVES GmbH & Co. KG | Location: Goldenstedt, Germany - 2023-07-24 *)
    M_DR_DIESEL_TECHNOLOGIES : UINT := 1381; (* Manufacturer: Dr. Diesel Technologies | Location: Murrieta, CA USA - 2023-07-24 *)
    M_THORNWAVE_LABS : UINT := 1382; (* Manufacturer: Thornwave Labs Inc. | Location: Youngsville, NC USA - 2023-07-24 *)
    M_ALPEGO : UINT := 1383; (* Manufacturer: Alpego S.p.A. | Location: Lonigo, Italy - 2023-07-24 *)
    M_TECNOSEAL_FOUNDRY_S_R_L : UINT := 1384; (* Manufacturer: Tecnoseal Foundry S.r.l. | Location: Grosseto, Italy - 2023-07-24 *)
    M_PRO_CHARGING_SYSTEMS : UINT := 1385; (* Manufacturer: Pro Charging Systems, LLC | Location: La Vergne, TN USA - 2023-07-24 *)
    M_SMART_EYE : UINT := 1386; (* Manufacturer: Smart Eye AB | Location: Gothenburg, Sweden - 2023-07-24 *)
    M_RADEL : UINT := 1387; (* Manufacturer: Radel (Pty) Ltd | Location: Olivedale, South Africa - 2023-07-31 *)
    M_NIRA_TECHNOLOGY : UINT := 1388; (* Manufacturer: Nira Technology | Location: Eskisehir, Turkey - 2023-08-15 *)
    M_EVEX : UINT := 1389; (* Manufacturer: EVEX Co., LTD | Location: Busan, Republic of Korea - 2023-08-23 *)
    M_FJ_DYNAMICS_INTERNATIONAL_LIMITED : UINT := 1390; (* Manufacturer: FJ Dynamics International Limited | Location: Shenzhen, China - 2023-08-23 *)
    M_ARIENSCO : UINT := 1391; (* Manufacturer: AriensCo | Location: Brillion, WI USA - 2023-08-29 *)
    M_PHOENIX_AMERICA : UINT := 1392; (* Manufacturer: Phoenix America LLC | Location: Fort Wayne, IN USA - 2023-08-29 *)
    M_POWERLAND_TECHNOLOGY : UINT := 1393; (* Manufacturer: Powerland Technology Inc | Location: Nanjing, China - 2023-08-29 *)
    M_ZHEJIANG_RUIXING_ELECTROMECHANICAL_TECHNOLOGY : UINT := 1394; (* Manufacturer: Zhejiang Ruixing Electromechanical Technology Co., Ltd. | Location: Zhejiang, China *)
    M_MLB_INDUSTRIAL : UINT := 1395; (* Manufacturer: MLB Industrial | Location: Arundel, QLD Australia - 2023-09-15 *)
    M_FAST_AG_SOLUTIONS : UINT := 1396; (* Manufacturer: Fast Ag Solutions, LLC | Location: Windom, MN USA - 2023-10-04 *)
    M_SAMASZ_SP_Z_O_O : UINT := 1397; (* Manufacturer: SaMASZ Sp. Z o.o. | Location: Zabludow, Poland - 2023-10-04 *)
    M_GOBIUS_SENSOR_TECHNOLOGY : UINT := 1398; (* Manufacturer: Gobius Sensor Technology AB | Location: Ellös, Sweden - 2023-10-12 *)
    M_HANS_BRANTNER_AND_SOHN_FAHRZEUGBAUGESELLSCHAFT_MBH : UINT := 1399; (* Manufacturer: Hans Brantner & Sohn Fahrzeugbaugesellschaft mbH | Location: Laa an der Thaya, *)
    M_IWN_AND : UINT := 1400; (* Manufacturer: IWN GmbH & Co. KG | Location: Bielefeld, Germany - 2023-10-12 *)
    M_ROM_COMMUNICATIONS : UINT := 1401; (* Manufacturer: ROM Communications Inc. | Location: Kelowna, BC Canada - 2023-10-12 *)
    M_COMNAV_TECHNOLOGY : UINT := 1402; (* Manufacturer: ComNav Technology Ltd. | Location: Shanghai, China - 2023-10-20 *)
    M_ARCO_MARINE : UINT := 1403; (* Manufacturer: Arco Marine | Location: Pensacola, FL USA - 2023-10-23 *)
    M_BRUSA_HYPOWER_AG : UINT := 1404; (* Manufacturer: BRUSA HyPower AG | Location: Buchs, Switzerland - 2023-10-31 *)
    M_TELIG_ELECTRONICS : UINT := 1405; (* Manufacturer: TELIG Electronics | Location: Passo Fundo, Brazil - 2023-11-03 *)
    M_LUMILEX_ALT_SRL : UINT := 1406; (* Manufacturer: Lumilex ALT SRL | Location: Baicoi, PH Romania - 2023-11-08 *)
    M_OPEN_AGRICULTURE : UINT := 1407; (* Manufacturer: Open-Agriculture | Location: Gescher, Germany - 2023-11-10 *)
    M_LENCO_MARINE : UINT := 1408; (* Manufacturer: Lenco Marine Inc. | Location: Stuart, FL USA - 2023-11-13 *)
    M_Z_ELEKTRONIKA_KFT : UINT := 1409; (* Manufacturer: Z Elektronika Kft. | Location: Pécs, Hungary - 2023-12-04 *)
    M_ALLAN_EQUIPMENT_MANUFACTURING : UINT := 1410; (* Manufacturer: Allan Equipment Manufacturing Ltd. | Location: York, PE Canada - 2023-12-04 *)
    M_SHANGHAI_HUACE_NAVIGATION_TECHNOLOGY : UINT := 1411; (* Manufacturer: Shanghai Huace Navigation Technology Ltd. | Location: Shanghai, China - 2023-12-04 *)
    M_NAOCONTROL_S_L : UINT := 1412; (* Manufacturer: Naocontrol S.L. | Location: A Coruña, Spain - 2023-12-20 *)
    M_OHNOH2O : UINT := 1413; (* Manufacturer: OHNOH2O LLC | Location: Lake Worth, FL USA - 2023-12-20 *)
    M_INTRACOM_DEFENSE : UINT := 1414; (* Manufacturer: INTRACOM DEFENSE S.A. | Location: Koropi, Greece - 2023-12-21 *)
    M_M_QUINAS_AGR_COLAS_JACTO : UINT := 1415; (* Manufacturer: Máquinas Agrícolas Jacto S.A. | Location: Pompéia, São Paulo, Brazil - 2024-01-04 *)
    M_WAVETRONIX : UINT := 1416; (* Manufacturer: Wavetronix LLC | Location: Springville, UT USA - 2024-01-04 *)
    M_REVATEK : UINT := 1417; (* Manufacturer: Revatek LLC | Location: Menomonee Falls, WI USA - 2024-01-07 *)
    M_KARLUNA_ENGINEERING : UINT := 1418; (* Manufacturer: Karluna Engineering | Location: İzmir, Turkey - 2024-01-07 *)
    M_IPATCH_MARINE : UINT := 1419; (* Manufacturer: iPatch Marine | Location: Camberwell, Australia - 2024-01-11 *)
    M_TALOS_PRECISION_MEASUREMENT_TECHNOLOGIES : UINT := 1420; (* Manufacturer: TALOS - Precision Measurement Technologies | Location: Clearwater, FL USA - *)
    M_CLARIOS : UINT := 1421; (* Manufacturer: Clarios, LLC | Location: Glendale, WI USA - 2024-01-11 *)
    M_XTCU_AG : UINT := 1422; (* Manufacturer: xTCU AG | Location: Vaduz, Liechtenstein - 2024-01-11 *)
    M_AC : UINT := 1423; (* Manufacturer: AC S.A. | Location: Bialystok, Poland - 2024-01-11 *)
    M_BEWIS : UINT := 1424; (* Manufacturer: Bewis | Location: Wuxi, China - 2024-05-07 *)
    M_ELECTRONICS_IN_AGRICULTURE_SCHOOL_OF_ENGINEERING_UNIVERSITY_OF_GALWAY : UINT := 1425; (* Manufacturer: Electronics in Agriculture, School of Engineering, University of Galway | Location: *)
    M_SAMSON_GROUP : UINT := 1426; (* Manufacturer: Samson Group | Location: Viborg, Denmark - 2024-02-01 *)
    M_REITER_RESPIRO : UINT := 1427; (* Manufacturer: REITER RESPIRO | Location: Hofkirchen an der Trattnach, Austria - 2024-02-11 *)
    M_SAMO_MASCHINENBAU : UINT := 1428; (* Manufacturer: Samo Maschinenbau GmbH | Location: Ottnang am Hausruck, Austria - 2024-02-12 *)
    M_NIKOLA : UINT := 1429; (* Manufacturer: Nikola Corporation | Location: Phoenix, AZ USA - 2024-02-13 *)
    M_MANTRACOURT_ELECTRONICS : UINT := 1430; (* Manufacturer: Mantracourt Electronics Ltd | Location: Exeter, Devon UK - 2024-02-13 *)
    M_NAUTO : UINT := 1431; (* Manufacturer: Nauto Inc. | Location: Sunnyvale, CA USA - 2024-03-13 *)
    M_MDH_DEFENCE : UINT := 1432; (* Manufacturer: MDH Defence Ltd. | Location: Amesbury, Wiltshire UK - 2024-03-13 *)
    M_UNICONTROL_APS : UINT := 1433; (* Manufacturer: Unicontrol ApS | Location: Odense, Denmark - 2024-03-13 *)
    M_ESURVEY_GNSS : UINT := 1434; (* Manufacturer: eSurvey GNSS Ltd. | Location: Shanghai, China - 2024-03-13 *)
    M_HEILONGJIANG_HUIDA_TECHNOLOGY : UINT := 1435; (* Manufacturer: Heilongjiang Huida Technology Co., Ltd | Location: Harbin, Hei long jiang, China - *)
    M_M_EXTEND : UINT := 1436; (* Manufacturer: M-extend | Location: Acigné, France - 2024-03-13 *)
    M_DOKEN_TECHNOLOGY : UINT := 1437; (* Manufacturer: DOKEN Technology Co. Ltd. | Location: Konya, Turkey - 2024-03-13 *)
    M_AEOLIONICS : UINT := 1438; (* Manufacturer: Aeolionics | Location: Mercer Island, WA USA - 2024-03-14 *)
    M_PREDICTWIND : UINT := 1439; (* Manufacturer: PredictWind Ltd | Location: Port England, Auckland, New Zealand - 2024-03-13 *)
    M_EGIS_MOBILE_ELECTRIC : UINT := 1440; (* Manufacturer: Egis Mobile Electric | Location: Bellingham, WA USA - 2024-03-14 *)
    M_SHANGHAI_ALLYNAV_TECHNOLOGY : UINT := 1441; (* Manufacturer: Shanghai Allynav Technology Co.,Ltd. | Location: Shanghai, China - 2024-03-14 *)
    M_EVYTRA : UINT := 1442; (* Manufacturer: EVYTRA GmbH | Location: Villingen-Schwenningen, BW, Germany - 2024-04-17 *)
    M_SOILESSENTIALS_LIMITED : UINT := 1443; (* Manufacturer: SoilEssentials Limited | Location: Brechin, Angus, UK - 2024-04-17 *)
    M_MICROPOWER_GROUP : UINT := 1444; (* Manufacturer: Micropower Group | Location: Växjö, Småland, Sweden - 2024-04-17 *)
    M_STARBOARD_YACHT_GROUP : UINT := 1445; (* Manufacturer: Starboard Yacht Group | Location: Dania Beach, FL - 2024-04-17 *)
    M_ROSWELL_MARINE : UINT := 1446; (* Manufacturer: Roswell Marine | Location: Rockledge, FL - 2024-04-17 *)
    M_INNOTAG_DISTRIBUTIONS : UINT := 1447; (* Manufacturer: Innotag Distributions Inc. | Location: Beloeil, Quebec, Canada - 2024-04-17 *)
    M_ELMER_S_MANUFACTURING : UINT := 1448; (* Manufacturer: Elmer's Manufacturing | Location: Altona, Manitoba, Canada - 2024-04-17 *)
    M_BONTAZ_CENTRE : UINT := 1449; (* Manufacturer: Bontaz Centre | Location: Marnaz, France - 2024-04-17 *)
    M_AGRIVAUX : UINT := 1450; (* Manufacturer: Agrivaux | Location: Charleroi, France - 2024-04-17 *)
    M_GUANGDONG_EPROPULSION_TECHNOLOGY : UINT := 1451; (* Manufacturer: Guangdong ePropulsion Technology Ltd. | Location: Guangdong Province, MD, China - *)
    M_MICRO_AIR : UINT := 1452; (* Manufacturer: Micro-Air LLC | Location: Hamilton, NJ USA - 2024-04-17 *)
    M_VITAL_BATTERY : UINT := 1453; (* Manufacturer: Vital Battery | Location: Taylors Beach, NSW, Australia - 2024-04-17 *)
    M_QTIS_B_V : UINT := 1454; (* Manufacturer: QTIS B.V. | Location: Sliedrecht, The Netherlands - 2024-05-07 *)
    M_EBERSP_CHER_CLIMATE_CONTROL_SYSTEMS_INTERNATIONAL : UINT := 1455; (* Manufacturer: Eberspächer Climate Control Systems International GmbH | Location: Esslingen, *)
    M_KRAMPE_FAHRZEUGBAU : UINT := 1456; (* Manufacturer: Krampe Fahrzeugbau GmbH | Location: Coesfeld, North Rhine Westphalia, Germany - *)
    M_ALBACH_MASCHINENBAU_AG : UINT := 1457; (* Manufacturer: Albach Maschinenbau AG | Location: Vohburg, Bayer, Germany - 2024-05-07 *)
    M_RIDECONTROLLER : UINT := 1458; (* Manufacturer: RideController LLC | Location: Kansas City, MO USA - 2024-06-14 *)
    M_ADVANCED_INPUT_SYSTEMS : UINT := 1459; (* Manufacturer: Advanced Input Systems | Location: Coeur d'Alene, ID USA - 2024-06-14 *)
    M_TOCARO_BLUE : UINT := 1460; (* Manufacturer: Tocaro Blue | Location: Pensacola, FL USA - 2024-06-14 *)
    M_VANQUISH_YACHTS : UINT := 1461; (* Manufacturer: Vanquish Yachts | Location: Marknesse, The Netherlands - 2024-06-14 *)
    M_TRACKUNIT_APS : UINT := 1462; (* Manufacturer: Trackunit ApS | Location: Aalborg, Denmark - 2024-06-14 *)
    M_STOK_ELECTRIC : UINT := 1463; (* Manufacturer: STOK Electric | Location: Lieshout, Noord-Brabant, The Netherlands - 2024-06-14 *)
    M_HI_TARGET_SURVEYING_INSTRUMENT : UINT := 1464; (* Manufacturer: Hi-Target Surveying Instrument Co., Ltd. | Location: Guangzhou, Guangdong, China - *)
    M_WATTECO : UINT := 1465; (* Manufacturer: Watteco | Location: Lanester, Brittany, France - 2024-07-01 *)
    M_SVEAVERKEN_SVEA_AGRI : UINT := 1466; (* Manufacturer: Sveaverken Svea Agri AB | Location: Katrineholm, Sweden - 2024-07-01 *)
    M_E_T_S_R_L : UINT := 1467; (* Manufacturer: S.A.E.T. s.r.l. | Location: Costigliole Saluzzo, Italy - 2024-07-01 *)
    M_SENQUIP : UINT := 1468; (* Manufacturer: Senquip | Location: Taylors Beach, NSW, Australia - 2024-08-02 *)
    M_LS_MTRON : UINT := 1469; (* Manufacturer: LS Mtron | Location: Wanju-gun, Jeollabuk-do, Republic of Korea - 2024-08-02 *)
    M_GEMONE_NV : UINT := 1470; (* Manufacturer: GemOne NV | Location: Waregem, Belgium - 2024-08-02 *)
    M_FT_TECHNOLOGIES : UINT := 1471; (* Manufacturer: FT Technologies | Location: Sunbury on Thames, UK - 2024-08-02 *)
    M_ACCULON_ENERGY : UINT := 1472; (* Manufacturer: Acculon Energy | Location: Columbus, OH USA - 2024-09-16 *)
    M_CRANESMART_SYSTEMS : UINT := 1473; (* Manufacturer: Cranesmart Systems, Inc. | Location: Edmonton, Alberta, Canada - 2024-09-16 *)
    M_CALEX_ELECTRONICS_LIMITED : UINT := 1474; (* Manufacturer: Calex Electronics Limited | Location: Leighton Buzzard, Bedfordshire, UK - *)
    M_DSP_SOLUTIONS : UINT := 1475; (* Manufacturer: DSP Solutions, Inc. | Location: Oxnard, CA USA - 2024-09-16 *)
    M_WILHELM_STOLL_MASCHINENFABRIK : UINT := 1476; (* Manufacturer: Wilhelm Stoll Maschinenfabrik GmbH | Location: Lengede, Germany - 2024-09-16 *)
    M_TOBROCO_GIANT : UINT := 1477; (* Manufacturer: TOBROCO-GIANT | Location: Oisterwijk, The Netherlands - 2024-09-16 *)
    M_ALPS_ALPINE : UINT := 1478; (* Manufacturer: Alps Alpine Co., Ltd. | Location: Tokyo, Japan - 2024-09-16 *)
    M_A_ELECTRONIX : UINT := 1479; (* Manufacturer: A-Electronix | Location: Nybrostrand, Skane, Sweden - 2024-09-16 *)
    M_THERMO_KING : UINT := 1480; (* Manufacturer: Thermo King | Location: Bloomington, MN USA - 2024-10-14 *)
    M_E_FORCE_MARINE : UINT := 1481; (* Manufacturer: E-Force Marine | Location: Miami Gardens, FL USA - 2024-10-14 *)
    M_CMC_MARINE : UINT := 1482; (* Manufacturer: CMC Marine | Location: Milano, Italy - 2024-10-14 *)
    M_NANJING_SANDEMARINE_INFORMATION_TECHNOLOGY : UINT := 1483; (* Manufacturer: Nanjing Sandemarine Information Technology Co., Ltd. | Location: Nanjing, Jiangsu *)
    M_AGROOSA : UINT := 1484; (* Manufacturer: AgroOSA | Location: Robakowo, WLKP, Poland - 2024-11-09 *)
    M_LESTER_ELECTRICAL : UINT := 1485; (* Manufacturer: Lester Electrical | Location: Lincoln, NE USA - 2024-11-09 *)
    M_XPANNER : UINT := 1486; (* Manufacturer: Xpanner | Location: Seoul, South Korea - 2024-11-09 *)
    M_GEOSOFT : UINT := 1487; (* Manufacturer: Geosoft | Location: Seoul, South Korea - 2024-11-09 *)
    M_BOETKIN_TECHNOLOGY : UINT := 1488; (* Manufacturer: Boetkin Technology Co., LTD | Location: Dongguan City, Guangdong Province, China - *)
    M_LITE_CHECK : UINT := 1489; (* Manufacturer: Lite-Check LLC | Location: Spokane, WA USA - 2024-11-09 *)
    M_CLEAN_REPUBLIC_SODO : UINT := 1490; (* Manufacturer: Clean Republic SODO, LLC | Location: Seattle, WA USA - 2024-11-09 *)
    M_POWER_POLLEN : UINT := 1491; (* Manufacturer: Power Pollen | Location: Ames, IA USA - 2024-11-09 *)
    M_SOFTIVERT : UINT := 1492; (* Manufacturer: Softivert | Location: Gabaston, France - 2024-11-09 *)
    M_JANTOP_OY : UINT := 1493; (* Manufacturer: Jantop Oy | Location: Vieremä, Finland - 2024-11-09 *)
    M_RAPITRONICS : UINT := 1494; (* Manufacturer: RAPITRONICS | Location: Makoszyn, Poland - 2025-01-09 *)
    M_FLYAGDATA : UINT := 1495; (* Manufacturer: FlyAgData | Location: Zielona Góra, Poland - 2025-01-06 *)
    M_AGRIROBOT : UINT := 1496; (* Manufacturer: AgriRobot | Location: Kongens Lyngby, Denmark - 2025-01-06 *)
    M_ERMO : UINT := 1497; (* Manufacturer: ERMO Spa | Location: Casalbuttano ed Uniti, Italy - 2025-01-06 *)
    M_PM_PFANZELT_MASCHINENBAU : UINT := 1498; (* Manufacturer: PM Pfanzelt Maschinenbau GmbH | Location: Rettenbach, Germany - 2025-01-06 *)
    M_HYDRASYSTEM_SP_Z_O_O : UINT := 1499; (* Manufacturer: Hydrasystem SP. Z O.O. | Location: Janki, Poland - 2025-01-06 *)
    M_SCANSTRUT : UINT := 1500; (* Manufacturer: Scanstrut Inc. | Location: Westbrook, CT USA - 2025-01-06 *)
    M_REVERSO_PUMPS : UINT := 1501; (* Manufacturer: Reverso Pumps LLC | Location: Davie, FL USA - 2025-01-06 *)
    M_BARANTECH : UINT := 1502; (* Manufacturer: Barantech | Location: Kiriyat Gat, Israel - 2025-01-06 *)
    M_ROSEMOUNT_SPECIALTY_PRODUCTS : UINT := 1503; (* Manufacturer: Rosemount Specialty Products | Location: East Wenatchee, WA USA - 2025-01-06 *)
    M_NIMBUS_POWER_SYSTEMS : UINT := 1504; (* Manufacturer: Nimbus Power Systems, Inc. | Location: Groton, CT USA - 2025-01-06 *)
    M_BC_MOTION : UINT := 1505; (* Manufacturer: BC Motion | Location: Saginaw, MN USA - 2025-01-06 *)
    M_EXPION360 : UINT := 1506; (* Manufacturer: Expion360 | Location: Redmond, OR USA - 2025-02-11 *)
    M_APEX_AI : UINT := 1507; (* Manufacturer: Apex.AI, Inc. | Location: Palo Alto, CA USA - 2025-02-11 *)
    M_XWATCH_SAFETY_SOLUTIONS_PART_OF_HEXAGON : UINT := 1508; (* Manufacturer: Xwatch Safety Solutions Ltd. part of Hexagon | Location: Three Legged Cross, *)
    M_BONDIOLI_AND_PAVESI_1509 : UINT := 1509; (* Manufacturer: Bondioli & Pavesi | Location: Suzzara, MN, Italy - 2025-02-11 *)
    M_AUSTIN_MOTOR_WORKS : UINT := 1510; (* Manufacturer: Austin Motor Works | Location: Austin, TX USA - 2025-02-11 *)
    M_APATOR_METRA_S_R_O : UINT := 1511; (* Manufacturer: APATOR METRA s.r.o. | Location: Sumperk, Czech Republic - 2025-02-11 *)
    M_LUMITEC : UINT := 1512; (* Manufacturer: Lumitec LLC | Location: Delray Beach, FL USA - 2025-02-11 *)
    M_SY_KLONE_INTERNATIONAL : UINT := 1513; (* Manufacturer: Sy-Klone International | Location: Jacksonville, FL USA - 2025-02-11 *)
    M_SYMX_AI : UINT := 1514; (* Manufacturer: SYMX.ai | Location: Sudbury, Ontario, Canada - 2025-02-11 *)
    M_INGENIER_A_Y_SISTEMAS_CEREA : UINT := 1515; (* Manufacturer: Ingeniería y Sistemas Cerea | Location: Valladolid, Castilla y León, Spain - *)
    M_THERMIS_SPOL_S_R_O : UINT := 1516; (* Manufacturer: THERMIS spol. s r.o. | Location: Brno, Czech Republic - 2025-02-11 *)
    M_DAEDONG : UINT := 1517; (* Manufacturer: Daedong Corporation | Location: Daegu, South Korea - 2025-02-11 *)
    M_NOVA_KOOL_MANUFACTURING_ULC : UINT := 1518; (* Manufacturer: Nova Kool Manufacturing ULC | Location: Coquitlam, BC, Canada - 2025-04-09 *)
    M_VOLBOFF_ELECTRON_SCIENCE_AND_TECHNOLOGY : UINT := 1519; (* Manufacturer: Volboff Electron Science and Technology Co., Ltd. | Location: Minhang District, *)
    M_SRT_MARINE_SYSTEMS_PLC : UINT := 1520; (* Manufacturer: SRT Marine Systems PLC | Location: Bath, UK - 2025-04-09 *)
    M_AGRICOLMECCANICA : UINT := 1521; (* Manufacturer: Agricolmeccanica | Location: Torviscosa, Udine, Italy - 2025-04-09 *)
    M_AMERICAN_THERMAL_INSTRUMENTS : UINT := 1522; (* Manufacturer: American Thermal Instruments | Location: Dayton, OH USA - 2025-04-09 *)
    M_CARLSON_SOFTWARE : UINT := 1523; (* Manufacturer: Carlson Software | Location: Maysville, KY USA - 2025-04-09 *)
    M_OCEAN_INFINITY_SOLUTIONS_LIMITED : UINT := 1524; (* Manufacturer: Ocean Infinity Solutions Limited | Location: London, UK - 2025-04-09 *)
    M_EMSISO_EMDRIVE : UINT := 1525; (* Manufacturer: Emsiso-emDrive | Location: Pesnica pri Mariboru, Slovenia - 2025-04-09 *)
    M_MITSUBISHI_MAHINDRA_AGRICULTURAL_MACHINERY : UINT := 1526; (* Manufacturer: MITSUBISHI MAHINDRA AGRICULTURAL MACHINERY CO.,LTD. | Location: Matsue, Shimane, *)
    M_RICHARDT_STEUER_UND_REGELGERAETE : UINT := 1527; (* Manufacturer: Richardt Steuer- und Regelgeraete GmbH | Location: Oberaula, Germany - 2025-04-09 *)
    M_SAVANT_TECHNOLOGY : UINT := 1528; (* Manufacturer: Savant Technology | Location: Casper, WY USA - 2025-04-09 *)
    M_INDUSTRIE_ELEKTRONIK_BRILON : UINT := 1529; (* Manufacturer: Industrie Elektronik Brilon GmbH | Location: Brilon, NRW, Germany - 2025-04-09 *)
    M_ROELAMA_B_V : UINT := 1530; (* Manufacturer: Roelama B.V. | Location: Alphen, Noord-Brabant, The Netherlands - 2025-04-09 *)
    M_KOBELCO_CONSTRUCTION_MACHINERY : UINT := 1531; (* Manufacturer: Kobelco Construction Machinery Co.,Ltd. | Location: Hiroshima, Japan - 2025-04-09 *)
    M_E_SWITCH : UINT := 1532; (* Manufacturer: E-Switch, Inc. | Location: Brooklyn Park, MN USA - 2025-04-09 *)
    M_RIEKER : UINT := 1533; (* Manufacturer: Rieker Inc. | Location: Aston, PA USA - 2025-04-09 *)
    M_BLUVEIN : UINT := 1534; (* Manufacturer: BluVein | Location: Northgate, Queensland, Australia - 2025-04-09 *)
    M_LOX_CONTAINER_TECHNOLOGY : UINT := 1535; (* Manufacturer: LOX Container Technology AB | Location: Stockholm, Sweden - 2025-04-09 *)
    M_TATRA_TRUCKS_A_S : UINT := 1536; (* Manufacturer: Tatra Trucks a.s. | Location: Koprivnice, Czech Republic - 2025-04-09 *)
    M_ANYLOAD_WEIGH_AND_MEASURE : UINT := 1537; (* Manufacturer: Anyload Weigh & Measure Inc. | Location: Bournaby, BC, Canada - 2025-04-25 *)
    M_QUICK : UINT := 1538; (* Manufacturer: Quick S.p.A. | Location: Piangipane - Ravenna, Italy - 2025-04-25 *)
    M_CEDAY_INFORMATION_TECHNOLOGIES : UINT := 1539; (* Manufacturer: Ceday Information Technologies | Location: Izmir, Bornova, Turkey - 2025-04-25 *)
    M_IDEAS_AND_MOTION : UINT := 1540; (* Manufacturer: Ideas & Motion | Location: Cherasco (CN), Italy - 2025-04-25 *)
    M_SOLID_STATE_MARINE : UINT := 1541; (* Manufacturer: Solid State Marine | Location: West Bridgewater, MA USA - 2025-04-25 *)
    M_GLOBAL_DIGITAL_INSTRUMENTS : UINT := 1542; (* Manufacturer: Global Digital Instruments | Location: Fairport, NY USA - 2025-04-25 *)
    M_GT_JOYSTICKS_AG : UINT := 1543; (* Manufacturer: GT Joysticks AG | Location: Bruegg, BE, Switzerland - 2025-04-25 *)
    M_GEOPHYSICAL_SURVEY_SYSTEMS : UINT := 1544; (* Manufacturer: Geophysical Survey Systems, Inc. | Location: Nashua, NH, USA - 2025-05-09 *)
    M_ROADEAZY : UINT := 1545; (* Manufacturer: RoadEazy | Location: Sunnyvale, CA USA - 2025-05-09 *)
    M_ESMART : UINT := 1546; (* Manufacturer: ESMART | Location: Indianapolis, IN USA - 2025-05-09 *)
    M_WEICHAI_LOVOL_INTELLIGENT_AGRICULTURAL_TECHNOLOGY : UINT := 1547; (* Manufacturer: Weichai Lovol Intelligent Agricultural Technology Co., Ltd. | Location: Weifang *)
    M_AM : UINT := 1549; (* Manufacturer: AM Co., Ltd. | Location: Gwacheon-si, Gyeonggi-do, South Korea - 2025-05-09 *)
    M_MARIO_TANZI : UINT := 1550; (* Manufacturer: Mario Tanzi S.A. | Location: Arequito, Santa Fe, Argentina - 2025-05-09 *)
    M_LMCE_GROUP : UINT := 1551; (* Manufacturer: LMCE Group | Location: Loimaa, Finland - 2025-05-09 *)
    M_ANTONIOSI_TECNOLOGIA_AGROINDUSTRIAL_LTDA : UINT := 1552; (* Manufacturer: Antoniosi Tecnologia Agroindustrial Ltda | Location: Matão, São Paulo, Brasil - *)
    M_BOUGHTON_ENGINEERING : UINT := 1553; (* Manufacturer: Boughton Engineering LTD | Location: Wolverhampton, West Midlands, UK - 2025-06-16 *)
    M_FRIGUS : UINT := 1554; (* Manufacturer: Frigus AB | Location: Gothenburg, Sweden - 2025-06-16 *)
    M_SAFIERY : UINT := 1555; (* Manufacturer: Safiery | Location: Arundel, Australia - 2025-06-16 *)
    M_B_KAUFMANN_AG_LANDMASCHINEN : UINT := 1556; (* Manufacturer: B. Kaufmann AG Landmaschinen | Location: 6246 Altishofen, Switzerland - 2025-06-16 *)
    M_INTERFACOM_U : UINT := 1557; (* Manufacturer: Interfacom S.A.U. | Location: Barcelona, Spain - 2025-06-16 *)
    M_INTANGLES_LAB_PRIVATE_LIMITED : UINT := 1558; (* Manufacturer: Intangles Lab Private Limited | Location: Pune, Maharashtra, India - 2025-06-16 *)
    M_KAR_TECH : UINT := 1559; (* Manufacturer: Kar-Tech, Inc. | Location: Delafield, WI, USA - 2025-06-16 *)
    M_MACOME : UINT := 1560; (* Manufacturer: MACOME CORPORATION | Location: Kami-ina, Nagano, Japan - 2025-06-16 *)
    M_FOX_MARINE : UINT := 1561; (* Manufacturer: Fox Marine | Location: Rising Sun, MD, USA - 2025-06-16 *)
    M_KINGSAT_COMMUNICATIONS : UINT := 1562; (* Manufacturer: Kingsat Communications Co., Ltd | Location: HuangGe Town, NanSha District, *)
    M_WABTEC_GRAHAM_WHITE : UINT := 1563; (* Manufacturer: Wabtec Graham White | Location: Salem, VA, USA - 2025-08-01 *)
    M_PRO_GUIDE_BATTERIES : UINT := 1564; (* Manufacturer: Pro-Guide Batteries | Location: Golden, MO, USA - 2025-08-01 *)
    M_LIVEMAC : UINT := 1565; (* Manufacturer: Livemac Co., Ltd. | Location: Jeonbuk, South Korea - 2025-08-01 *)
    M_OUTSET : UINT := 1566; (* Manufacturer: OUTSET | Location: Sandrigo, Vicenza, Italy - 2025-08-01 *)
    M_HAGEDORN_SOFTWARE_ENGINEERING : UINT := 1567; (* Manufacturer: Hagedorn Software Engineering GmbH | Location: Warendorf, Germany - 2025-08-01 *)
    M_AIGRO : UINT := 1568; (* Manufacturer: Aigro | Location: Best, Noord-Brabant, The Netherlands - 2025-08-01 *)
    M_621_TECHNOLOGIES : UINT := 1569; (* Manufacturer: 621 Technologies Inc. | Location: Petrolia, ON Canada - 2019-10-02 *)
    M_UNVERFERTH_MANUFACTURING_COMPANY : UINT := 1570; (* Manufacturer: Unverferth Manufacturing Company Inc. | Location: Kalida, OH, USA - 2025-08-01 *)
    M_SUPER_B : UINT := 1571; (* Manufacturer: Super B | Location: Hengelo, Overijssel, Netherlands - 2025-08-01 *)
    M_SMARTLINE : UINT := 1572; (* Manufacturer: SMARTLINE Co., Ltd. | Location: Seoul, South Korea - 2025-08-01 *)
    M_R_H_SHEPPARD : UINT := 1573; (* Manufacturer: R.H. Sheppard | Location: Hanover, PA, USA - 2025-08-04 *)
    M_SIGMA4_SRL : UINT := 1574; (* Manufacturer: SIGMA4 SRL | Location: Russi, Italy - 2025-08-12 *)
    M_DIESELHEAT : UINT := 1575; (* Manufacturer: DieselHeat | Location: Cygnet, Tasmania, Australia - 2025-08-12 *)
    M_RB_INTERNATIONAL_S_R_L : UINT := 1576; (* Manufacturer: RB International S.r.l. | Location: Città Di Castello, Italy - 2025-08-12 *)
    M_IRONSTONE_AG : UINT := 1577; (* Manufacturer: Ironstone AG | Location: Toodyay, WA, Australia - 2025-08-12 *)
    M_MIDNITE_SOLAR : UINT := 1578; (* Manufacturer: MidNite Solar Inc. | Location: Arlington, WA, USA - 2025-09-11 *)
    M_HYDRO_ENGINEERING : UINT := 1579; (* Manufacturer: Hydro Engineering | Location: Norwood Young America, MN, USA - 2025-09-11 *)
    M_NABTESCO : UINT := 1580; (* Manufacturer: Nabtesco Corporation | Location: Tokyo, Japan - 2025-09-11 *)
    M_METRO_MARINE : UINT := 1581; (* Manufacturer: Metro Marine LLC | Location: Englewood NJ, USA - 2025-09-11 *)
    M_SAMSUNG_HEAVY_INDUSTRIES : UINT := 1582; (* Manufacturer: Samsung Heavy Industries Co., Ltd. | Location: Seongnam-si, Gyeongi-do, South Korea *)
    M_MULTI_WING_GROUP : UINT := 1583; (* Manufacturer: MULTI-WING GROUP A/S | Location: Vedbæk, Denmark - 2025-10-30 *)
    M_TWK_ELEKTRONIK : UINT := 1584; (* Manufacturer: TWK-ELEKTRONIK GmbH | Location: Düsseldorf, NRW, Germany - 2025-09-11 *)
    M_QIANXUN_SPATIAL_INTELLIGENCE : UINT := 1585; (* Manufacturer: Qianxun Spatial Intelligence (Zhejiang) Inc. | Location: Zhejiang, China - *)
    M_XAG : UINT := 1586; (* Manufacturer: XAG CO., LTD. | Location: Guangzhou, Guangdong, China - 2025-09-11 *)
    M_BURGER_GROUP : UINT := 1587; (* Manufacturer: BURGER GROUP | Location: Schonach, Baden-Wuerttemberg, Germany - 2025-09-11 *)
    M_MORESIL : UINT := 1588; (* Manufacturer: MORESIL | Location: Posadas, Spain - 2025-10-30 *)
    M_H_BNER_AND : UINT := 1589; (* Manufacturer: HÜBNER GmbH & Co. KG | Location: Kassel, Germany - 2025-10-30 *)
    M_MONPAINEIS : UINT := 1590; (* Manufacturer: Monpaineis | Location: São Paulo, Brasil - 2025-10-30 *)
    M_WATERWORLD_ELECTRONICS : UINT := 1591; (* Manufacturer: WaterWorld Electronics | Location: Oldemarkt, The Netherlands - 2025-10-30 *)
    M_INCOMAGRI_M_QUINAS_AGR_COLAS_LTDA : UINT := 1592; (* Manufacturer: Incomagri Máquinas Agrícolas Ltda | Location: Itapira, Brazil - 2025-10-30 *)
    M_CORDON_TECHNOLOGIES : UINT := 1593; (* Manufacturer: Cordon Technologies | Location: Maidenhead, Berkshire, UK - 2025-10-30 *)
    M_ELWELL : UINT := 1594; (* Manufacturer: Elwell Corporation | Location: Washougal, WA, USA - 2025-10-30 *)
    M_PRUEFREX_ENGINEERING_E_MOTION : UINT := 1595; (* Manufacturer: Pruefrex engineering e motion gmbh | Location: Cadolzburg, Bayern, Germany - *)
    M_NEOSENS : UINT := 1596; (* Manufacturer: Neosens | Location: Pfaffenhofen an der Ilm, Bavaria, Germany - 2025-10-30 *)
    M_S_DESVOYS_AND_FILS : UINT := 1597; (* Manufacturer: S.A.S. Desvoys & Fils | Location: Landivy, Pays de la Loire, France - 2025-10-30 *)
    M_DI_GORO : UINT := 1598; (* Manufacturer: Di Goro | Location: Herston, QLD, Australia - 2025-10-30 *)
    M_KAMTEC : UINT := 1599; (* Manufacturer: Kamtec | Location: Jincheon-gun, Chungcheongbuk-do, Republic of Korea - 2025-10-30 *)
    M_CONSOLIDATED_METCO : UINT := 1600; (* Manufacturer: Consolidated Metco, Inc. | Location: Vancouver, WA, USA - 2025-10-30 *)
    M_T_CCI_MANUFACTURING : UINT := 1601; (* Manufacturer: T/CCI Manufacturing, LLC | Location: Decatur, IL, USA - 2026-01-27 *)
    M_NORCROSS_MARINE_PRODUCTS : UINT := 1602; (* Manufacturer: Norcross Marine Products | Location: Orlando, Florida, USA - 2026-01-27 *)
    M_ROCKVILLE_AUDIO : UINT := 1603; (* Manufacturer: Rockville Audio | Location: Inwood, NY, USA - 2025-12-08 *)
    M_ROVERSENSE_TECHNOLOGIES : UINT := 1604; (* Manufacturer: RoverSense Technologies | Location: McKinney, TX, USA - 2025-12-08 *)
    M_BLUE_WOLF : UINT := 1605; (* Manufacturer: Blue Wolf | Location: Garden City, ID, USA - 2025-12-08 *)
    M_SENSAR_MARINE : UINT := 1606; (* Manufacturer: SENSAR MARINE INC. | Location: Lexington, MA, USA - 2025-12-08 *)
    M_MICRO_KEY : UINT := 1607; (* Manufacturer: Micro-Key | Location: Leek, Groningen, The Netherlands - 2025-12-08 *)
    M_QUECTEL : UINT := 1608; (* Manufacturer: Quectel | Location: Shanghai, China - 2025-12-08 *)
    M_NANONORD : UINT := 1609; (* Manufacturer: NanoNord A/S | Location: Aalborg, Denmark - 2025-12-08 *)
    M_SIMARINE_D_O_O : UINT := 1610; (* Manufacturer: Simarine d.o.o. | Location: Maribor, Slovenia - 2025-12-08 *)
    M_NINGBO_HAIBO_GROUP : UINT := 1611; (* Manufacturer: Ningbo Haibo Group Co., Ltd. | Location: Ningbo, Zhejiang, China - 2025-12-08 *)
    M_BLUETTI : UINT := 1612; (* Manufacturer: BLUETTI | Location: Shenzhen, Guangdong, China - 2025-12-08 *)
    M_WHISPERPOWER : UINT := 1613; (* Manufacturer: Whisperpower | Location: Drachten, The Netherlands - 2025-12-08 *)
    M_RISSEEUW_TECHNIEK : UINT := 1614; (* Manufacturer: Risseeuw Techniek | Location: Schoondijke, The Netherlands - 2025-12-08 *)
    M_J_ASSY : UINT := 1615; (* Manufacturer: J.Assy | Location: Caldas Novas, Brazil - 2025-12-08 *)
    M_SATEL_OY : UINT := 1616; (* Manufacturer: Satel Oy | Location: Salo, Finland - 2025-12-08 *)
    M_DRUDLES_S_R_O : UINT := 1617; (* Manufacturer: DRUDLES s.r.o. | Location: Chocen, Czechia - 2025-12-08 *)
    M_THE_CARLISLE_AND_FINCH : UINT := 1618; (* Manufacturer: The Carlisle and Finch Co. | Location: Cincinnati, OH, USA - 2026-01-27 *)
    M_CLEMENS_AND : UINT := 1619; (* Manufacturer: Clemens GmbH & Co. KG | Location: Wittlich, Germany - 2026-01-27 *)
    M_BLUENAV_1620 : UINT := 1620; (* Manufacturer: BlueNav | Location: Arcachon, France - 2026-01-27 *)
    M_MACH : UINT := 1621; (* Manufacturer: Mach Inc. | Location: Finksburg, MD, USA - 2026-01-27 *)
    M_BRETTMEISTER_ELEKTRONIK : UINT := 1622; (* Manufacturer: Brettmeister Elektronik | Location: Paar, Germany - 2026-01-27 *)
    M_PRO_CHARGING_SYSTEMS_1623 : UINT := 1623; (* Manufacturer: PRO Charging Systems, LLC | Location: La Vergne, TN, USA - 2026-01-27 *)
